	VAR jointtarget CDP_1949 := [[-13.97, 36.67, 4.6, 0, 48.73, -199.13], [9E9, 9E9, 9E9, 9E9, 9E9, 9E9]];
	VAR jointtarget CDP_1950 := [[-13.99, 36.53, 4.84, 0, 48.63, -188.83], [9E9, 9E9, 9E9, 9E9, 9E9, 9E9]];
	VAR jointtarget CDP_1951 := [[-13.98, 36.39, 5.09, 0, 48.52, -178.5], [9E9, 9E9, 9E9, 9E9, 9E9, 9E9]];
	VAR jointtarget CDP_1952 := [[-13.96, 36.25, 5.33, 0, 48.42, -168.15], [9E9, 9E9, 9E9, 9E9, 9E9, 9E9]];
	VAR jointtarget CDP_1953 := [[-13.91, 36.12, 5.55, 0, 48.33, -157.77], [9E9, 9E9, 9E9, 9E9, 9E9, 9E9]];
	VAR jointtarget CDP_1954 := [[-13.84, 36, 5.76, 0, 48.24, -147.38], [9E9, 9E9, 9E9, 9E9, 9E9, 9E9]];
	VAR jointtarget CDP_1955 := [[-13.75, 35.89, 5.94, 0, 48.17, -136.97], [9E9, 9E9, 9E9, 9E9, 9E9, 9E9]];
	VAR jointtarget CDP_1956 := [[-13.64, 35.81, 6.08, 0, 48.11, -126.54], [9E9, 9E9, 9E9, 9E9, 9E9, 9E9]];
	VAR jointtarget CDP_1957 := [[-13.52, 35.74, 6.19, 0, 48.06, -116.09], [9E9, 9E9, 9E9, 9E9, 9E9, 9E9]];
	VAR jointtarget CDP_1958 := [[-13.4, 35.71, 6.26, 0, 48.04, -105.64], [9E9, 9E9, 9E9, 9E9, 9E9, 9E9]];
	VAR jointtarget CDP_1959 := [[-13.27, 35.69, 6.28, 0, 48.03, -95.19], [9E9, 9E9, 9E9, 9E9, 9E9, 9E9]];
	VAR jointtarget CDP_1960 := [[-13.2, 35.69, 6.28, 0, 48.03, -89.96], [9E9, 9E9, 9E9, 9E9, 9E9, 9E9]];
	VAR jointtarget CDP_1961 := [[-13.13, 35.69, 6.28, 0, 48.03, -89.89], [9E9, 9E9, 9E9, 9E9, 9E9, 9E9]];
	VAR jointtarget CDP_1962 := [[-13.06, 35.69, 6.28, 0, 48.03, -89.82], [9E9, 9E9, 9E9, 9E9, 9E9, 9E9]];
	VAR jointtarget CDP_1963 := [[-12.99, 35.69, 6.28, 0, 48.03, -89.75], [9E9, 9E9, 9E9, 9E9, 9E9, 9E9]];
	VAR jointtarget CDP_1964 := [[-12.93, 35.69, 6.28, 0, 48.03, -89.69], [9E9, 9E9, 9E9, 9E9, 9E9, 9E9]];
	VAR jointtarget CDP_1965 := [[-12.86, 35.69, 6.28, 0, 48.03, -89.62], [9E9, 9E9, 9E9, 9E9, 9E9, 9E9]];
	VAR jointtarget CDP_1966 := [[-12.79, 35.69, 6.28, 0, 48.03, -89.55], [9E9, 9E9, 9E9, 9E9, 9E9, 9E9]];
	VAR jointtarget CDP_1967 := [[-12.72, 35.69, 6.28, 0, 48.03, -89.48], [9E9, 9E9, 9E9, 9E9, 9E9, 9E9]];
	VAR jointtarget CDP_1968 := [[-12.65, 35.69, 6.27, 0, 48.03, -89.41], [9E9, 9E9, 9E9, 9E9, 9E9, 9E9]];
	VAR jointtarget CDP_1969 := [[-12.59, 35.69, 6.27, 0, 48.04, -89.35], [9E9, 9E9, 9E9, 9E9, 9E9, 9E9]];
	VAR jointtarget CDP_1970 := [[-12.52, 35.69, 6.27, 0, 48.04, -89.28], [9E9, 9E9, 9E9, 9E9, 9E9, 9E9]];
	VAR jointtarget CDP_1971 := [[-12.45, 35.69, 6.27, 0, 48.04, -89.21], [9E9, 9E9, 9E9, 9E9, 9E9, 9E9]];
	VAR jointtarget CDP_1972 := [[-12.38, 35.69, 6.27, 0, 48.04, -89.14], [9E9, 9E9, 9E9, 9E9, 9E9, 9E9]];
	VAR jointtarget CDP_1973 := [[-12.32, 35.69, 6.27, 0, 48.04, -89.07], [9E9, 9E9, 9E9, 9E9, 9E9, 9E9]];
	VAR jointtarget CDP_1974 := [[-12.25, 35.69, 6.26, 0, 48.04, -89.01], [9E9, 9E9, 9E9, 9E9, 9E9, 9E9]];
	VAR jointtarget CDP_1975 := [[-12.18, 35.69, 6.26, 0, 48.04, -88.94], [9E9, 9E9, 9E9, 9E9, 9E9, 9E9]];
	VAR jointtarget CDP_1976 := [[-12.11, 35.7, 6.26, 0, 48.05, -88.87], [9E9, 9E9, 9E9, 9E9, 9E9, 9E9]];
	VAR jointtarget CDP_1977 := [[-12.04, 35.7, 6.26, 0, 48.05, -88.8], [9E9, 9E9, 9E9, 9E9, 9E9, 9E9]];
	VAR jointtarget CDP_1978 := [[-11.98, 35.7, 6.25, 0, 48.05, -88.74], [9E9, 9E9, 9E9, 9E9, 9E9, 9E9]];
	VAR jointtarget CDP_1979 := [[-11.91, 35.7, 6.25, 0, 48.05, -88.67], [9E9, 9E9, 9E9, 9E9, 9E9, 9E9]];
	VAR jointtarget CDP_1980 := [[-11.89, 35.7, 6.25, 0, 48.05, -88.98], [9E9, 9E9, 9E9, 9E9, 9E9, 9E9]];
	VAR jointtarget CDP_1981 := [[-11.87, 35.7, 6.25, 0, 48.05, -89.63], [9E9, 9E9, 9E9, 9E9, 9E9, 9E9]];
	VAR jointtarget CDP_1982 := [[-11.86, 35.7, 6.25, 0, 48.05, -90.27], [9E9, 9E9, 9E9, 9E9, 9E9, 9E9]];
	VAR jointtarget CDP_1983 := [[-11.84, 35.7, 6.25, 0, 48.05, -90.92], [9E9, 9E9, 9E9, 9E9, 9E9, 9E9]];
	VAR jointtarget CDP_1984 := [[-11.82, 35.7, 6.25, 0, 48.05, -91.56], [9E9, 9E9, 9E9, 9E9, 9E9, 9E9]];
	VAR jointtarget CDP_1985 := [[-11.81, 35.7, 6.25, 0, 48.05, -92.21], [9E9, 9E9, 9E9, 9E9, 9E9, 9E9]];
	VAR jointtarget CDP_1986 := [[-11.79, 35.7, 6.25, 0, 48.05, -92.85], [9E9, 9E9, 9E9, 9E9, 9E9, 9E9]];
	VAR jointtarget CDP_1987 := [[-11.77, 35.69, 6.25, 0, 48.05, -93.5], [9E9, 9E9, 9E9, 9E9, 9E9, 9E9]];
	VAR jointtarget CDP_1988 := [[-11.76, 35.69, 6.26, 0, 48.05, -94.14], [9E9, 9E9, 9E9, 9E9, 9E9, 9E9]];
	VAR jointtarget CDP_1989 := [[-11.74, 35.69, 6.26, 0, 48.05, -94.79], [9E9, 9E9, 9E9, 9E9, 9E9, 9E9]];
	VAR jointtarget CDP_1990 := [[-11.72, 35.69, 6.26, 0, 48.05, -95.43], [9E9, 9E9, 9E9, 9E9, 9E9, 9E9]];
	VAR jointtarget CDP_1991 := [[-11.71, 35.69, 6.27, 0, 48.05, -96.08], [9E9, 9E9, 9E9, 9E9, 9E9, 9E9]];
	VAR jointtarget CDP_1992 := [[-11.69, 35.69, 6.27, 0, 48.05, -96.72], [9E9, 9E9, 9E9, 9E9, 9E9, 9E9]];
	VAR jointtarget CDP_1993 := [[-11.67, 35.68, 6.27, 0, 48.04, -97.37], [9E9, 9E9, 9E9, 9E9, 9E9, 9E9]];
	VAR jointtarget CDP_1994 := [[-11.66, 35.68, 6.28, 0, 48.04, -98.01], [9E9, 9E9, 9E9, 9E9, 9E9, 9E9]];
	VAR jointtarget CDP_1995 := [[-11.64, 35.68, 6.28, 0, 48.04, -98.66], [9E9, 9E9, 9E9, 9E9, 9E9, 9E9]];
	VAR jointtarget CDP_1996 := [[-11.62, 35.67, 6.29, 0, 48.04, -99.31], [9E9, 9E9, 9E9, 9E9, 9E9, 9E9]];
	VAR jointtarget CDP_1997 := [[-11.61, 35.67, 6.29, 0, 48.04, -99.95], [9E9, 9E9, 9E9, 9E9, 9E9, 9E9]];
	VAR jointtarget CDP_1998 := [[-11.59, 35.67, 6.3, 0, 48.03, -100.6], [9E9, 9E9, 9E9, 9E9, 9E9, 9E9]];
	VAR jointtarget CDP_1999 := [[-11.57, 35.66, 6.3, 0, 48.03, -101.24], [9E9, 9E9, 9E9, 9E9, 9E9, 9E9]];
	VAR jointtarget CDP_2000 := [[-10.48, 35.44, 6.7, 0, 47.87, -100.48], [9E9, 9E9, 9E9, 9E9, 9E9, 9E9]];
	VAR jointtarget CDP_2001 := [[-9.38, 35.23, 7.05, 0, 47.72, -99.38], [9E9, 9E9, 9E9, 9E9, 9E9, 9E9]];
	VAR jointtarget CDP_2002 := [[-8.27, 35.05, 7.36, 0, 47.59, -98.27], [9E9, 9E9, 9E9, 9E9, 9E9, 9E9]];
	VAR jointtarget CDP_2003 := [[-7.15, 34.89, 7.63, 0, 47.48, -97.15], [9E9, 9E9, 9E9, 9E9, 9E9, 9E9]];
	VAR jointtarget CDP_2004 := [[-6.03, 34.75, 7.87, 0, 47.38, -96.03], [9E9, 9E9, 9E9, 9E9, 9E9, 9E9]];
	VAR jointtarget CDP_2005 := [[-4.9, 34.64, 8.06, 0, 47.31, -94.9], [9E9, 9E9, 9E9, 9E9, 9E9, 9E9]];
	VAR jointtarget CDP_2006 := [[-3.77, 34.55, 8.21, 0, 47.24, -93.77], [9E9, 9E9, 9E9, 9E9, 9E9, 9E9]];
	VAR jointtarget CDP_2007 := [[-2.64, 34.48, 8.32, 0, 47.2, -92.64], [9E9, 9E9, 9E9, 9E9, 9E9, 9E9]];
	VAR jointtarget CDP_2008 := [[-1.51, 34.44, 8.4, 0, 47.17, -91.51], [9E9, 9E9, 9E9, 9E9, 9E9, 9E9]];
	VAR jointtarget CDP_2009 := [[-0.37, 34.42, 8.43, 0, 47.15, -90.37], [9E9, 9E9, 9E9, 9E9, 9E9, 9E9]];
	VAR jointtarget CDP_2010 := [[0.76, 34.42, 8.42, 0, 47.15, -89.24], [9E9, 9E9, 9E9, 9E9, 9E9, 9E9]];
	VAR jointtarget CDP_2011 := [[1.9, 34.45, 8.38, 0, 47.17, -88.1], [9E9, 9E9, 9E9, 9E9, 9E9, 9E9]];
	VAR jointtarget CDP_2012 := [[3.03, 34.5, 8.29, 0, 47.21, -86.97], [9E9, 9E9, 9E9, 9E9, 9E9, 9E9]];
	VAR jointtarget CDP_2013 := [[4.16, 34.57, 8.16, 0, 47.26, -85.84], [9E9, 9E9, 9E9, 9E9, 9E9, 9E9]];
	VAR jointtarget CDP_2014 := [[5.29, 34.67, 8, 0, 47.33, -84.71], [9E9, 9E9, 9E9, 9E9, 9E9, 9E9]];
	VAR jointtarget CDP_2015 := [[6.42, 34.79, 7.79, 0, 47.42, -83.58], [9E9, 9E9, 9E9, 9E9, 9E9, 9E9]];
	VAR jointtarget CDP_2016 := [[7.54, 34.94, 7.54, 0, 47.52, -82.46], [9E9, 9E9, 9E9, 9E9, 9E9, 9E9]];
	VAR jointtarget CDP_2017 := [[8.65, 35.11, 7.26, 0, 47.64, -81.35], [9E9, 9E9, 9E9, 9E9, 9E9, 9E9]];
	VAR jointtarget CDP_2018 := [[9.76, 35.3, 6.93, 0, 47.77, -80.24], [9E9, 9E9, 9E9, 9E9, 9E9, 9E9]];
	VAR jointtarget CDP_2019 := [[10.86, 35.51, 6.57, 0, 47.92, -79.14], [9E9, 9E9, 9E9, 9E9, 9E9, 9E9]];
	VAR jointtarget CDP_2020 := [[10.87, 35.52, 6.56, 0, 47.92, -79.46], [9E9, 9E9, 9E9, 9E9, 9E9, 9E9]];
	VAR jointtarget CDP_2021 := [[10.89, 35.52, 6.55, 0, 47.93, -80.1], [9E9, 9E9, 9E9, 9E9, 9E9, 9E9]];
	VAR jointtarget CDP_2022 := [[10.91, 35.52, 6.55, 0, 47.93, -80.75], [9E9, 9E9, 9E9, 9E9, 9E9, 9E9]];
	VAR jointtarget CDP_2023 := [[10.92, 35.52, 6.55, 0, 47.93, -81.39], [9E9, 9E9, 9E9, 9E9, 9E9, 9E9]];
	VAR jointtarget CDP_2024 := [[10.94, 35.53, 6.54, 0, 47.93, -82.04], [9E9, 9E9, 9E9, 9E9, 9E9, 9E9]];
	VAR jointtarget CDP_2025 := [[10.96, 35.53, 6.54, 0, 47.93, -82.68], [9E9, 9E9, 9E9, 9E9, 9E9, 9E9]];
	VAR jointtarget CDP_2026 := [[10.97, 35.53, 6.53, 0, 47.94, -83.33], [9E9, 9E9, 9E9, 9E9, 9E9, 9E9]];
	VAR jointtarget CDP_2027 := [[10.99, 35.53, 6.53, 0, 47.94, -83.97], [9E9, 9E9, 9E9, 9E9, 9E9, 9E9]];
	VAR jointtarget CDP_2028 := [[11.01, 35.53, 6.53, 0, 47.94, -84.62], [9E9, 9E9, 9E9, 9E9, 9E9, 9E9]];
	VAR jointtarget CDP_2029 := [[11.02, 35.54, 6.52, 0, 47.94, -85.27], [9E9, 9E9, 9E9, 9E9, 9E9, 9E9]];
	VAR jointtarget CDP_2030 := [[11.04, 35.54, 6.52, 0, 47.94, -85.91], [9E9, 9E9, 9E9, 9E9, 9E9, 9E9]];
	VAR jointtarget CDP_2031 := [[11.06, 35.54, 6.52, 0, 47.94, -86.56], [9E9, 9E9, 9E9, 9E9, 9E9, 9E9]];
	VAR jointtarget CDP_2032 := [[11.07, 35.54, 6.52, 0, 47.94, -87.2], [9E9, 9E9, 9E9, 9E9, 9E9, 9E9]];
	VAR jointtarget CDP_2033 := [[11.09, 35.54, 6.52, 0, 47.94, -87.85], [9E9, 9E9, 9E9, 9E9, 9E9, 9E9]];
	VAR jointtarget CDP_2034 := [[11.11, 35.54, 6.52, 0, 47.94, -88.49], [9E9, 9E9, 9E9, 9E9, 9E9, 9E9]];
	VAR jointtarget CDP_2035 := [[11.13, 35.54, 6.52, 0, 47.94, -89.14], [9E9, 9E9, 9E9, 9E9, 9E9, 9E9]];
	VAR jointtarget CDP_2036 := [[11.14, 35.54, 6.52, 0, 47.94, -89.78], [9E9, 9E9, 9E9, 9E9, 9E9, 9E9]];
	VAR jointtarget CDP_2037 := [[11.16, 35.54, 6.52, 0, 47.94, -90.43], [9E9, 9E9, 9E9, 9E9, 9E9, 9E9]];
	VAR jointtarget CDP_2038 := [[11.18, 35.54, 6.52, 0, 47.94, -91.07], [9E9, 9E9, 9E9, 9E9, 9E9, 9E9]];
	VAR jointtarget CDP_2039 := [[11.19, 35.54, 6.52, 0, 47.94, -91.72], [9E9, 9E9, 9E9, 9E9, 9E9, 9E9]];
	VAR jointtarget CDP_2040 := [[11.26, 35.54, 6.52, 0, 47.94, -91.98], [9E9, 9E9, 9E9, 9E9, 9E9, 9E9]];
	VAR jointtarget CDP_2041 := [[11.33, 35.53, 6.53, 0, 47.94, -91.91], [9E9, 9E9, 9E9, 9E9, 9E9, 9E9]];
	VAR jointtarget CDP_2042 := [[11.4, 35.53, 6.53, 0, 47.94, -91.84], [9E9, 9E9, 9E9, 9E9, 9E9, 9E9]];
	VAR jointtarget CDP_2043 := [[11.47, 35.53, 6.53, 0, 47.94, -91.78], [9E9, 9E9, 9E9, 9E9, 9E9, 9E9]];
	VAR jointtarget CDP_2044 := [[11.53, 35.53, 6.54, 0, 47.93, -91.71], [9E9, 9E9, 9E9, 9E9, 9E9, 9E9]];
	VAR jointtarget CDP_2045 := [[11.6, 35.53, 6.54, 0, 47.93, -91.64], [9E9, 9E9, 9E9, 9E9, 9E9, 9E9]];
	VAR jointtarget CDP_2046 := [[11.67, 35.52, 6.55, 0, 47.93, -91.57], [9E9, 9E9, 9E9, 9E9, 9E9, 9E9]];
	VAR jointtarget CDP_2047 := [[11.74, 35.52, 6.55, 0, 47.93, -91.5], [9E9, 9E9, 9E9, 9E9, 9E9, 9E9]];
	VAR jointtarget CDP_2048 := [[11.81, 35.52, 6.55, 0, 47.93, -91.44], [9E9, 9E9, 9E9, 9E9, 9E9, 9E9]];
	VAR jointtarget CDP_2049 := [[11.87, 35.52, 6.56, 0, 47.93, -91.37], [9E9, 9E9, 9E9, 9E9, 9E9, 9E9]];
	VAR jointtarget CDP_2050 := [[11.94, 35.52, 6.56, 0, 47.93, -91.3], [9E9, 9E9, 9E9, 9E9, 9E9, 9E9]];
	VAR jointtarget CDP_2051 := [[12.01, 35.51, 6.56, 0, 47.92, -91.23], [9E9, 9E9, 9E9, 9E9, 9E9, 9E9]];
	VAR jointtarget CDP_2052 := [[12.08, 35.51, 6.56, 0, 47.92, -91.16], [9E9, 9E9, 9E9, 9E9, 9E9, 9E9]];
	VAR jointtarget CDP_2053 := [[12.15, 35.51, 6.57, 0, 47.92, -91.09], [9E9, 9E9, 9E9, 9E9, 9E9, 9E9]];
	VAR jointtarget CDP_2054 := [[12.21, 35.51, 6.57, 0, 47.92, -91.03], [9E9, 9E9, 9E9, 9E9, 9E9, 9E9]];
	VAR jointtarget CDP_2055 := [[12.28, 35.51, 6.57, 0, 47.92, -90.96], [9E9, 9E9, 9E9, 9E9, 9E9, 9E9]];
	VAR jointtarget CDP_2056 := [[12.35, 35.51, 6.57, 0, 47.92, -90.89], [9E9, 9E9, 9E9, 9E9, 9E9, 9E9]];
	VAR jointtarget CDP_2057 := [[12.42, 35.51, 6.57, 0, 47.92, -90.82], [9E9, 9E9, 9E9, 9E9, 9E9, 9E9]];
	VAR jointtarget CDP_2058 := [[12.49, 35.51, 6.58, 0, 47.92, -90.75], [9E9, 9E9, 9E9, 9E9, 9E9, 9E9]];
	VAR jointtarget CDP_2059 := [[12.55, 35.5, 6.58, 0, 47.92, -90.69], [9E9, 9E9, 9E9, 9E9, 9E9, 9E9]];
	VAR jointtarget CDP_2060 := [[12.69, 35.52, 6.56, 0, 47.93, -85.39], [9E9, 9E9, 9E9, 9E9, 9E9, 9E9]];
	VAR jointtarget CDP_2061 := [[12.81, 35.55, 6.5, 0, 47.95, -74.94], [9E9, 9E9, 9E9, 9E9, 9E9, 9E9]];
	VAR jointtarget CDP_2062 := [[12.93, 35.61, 6.39, 0, 47.99, -64.5], [9E9, 9E9, 9E9, 9E9, 9E9, 9E9]];
	VAR jointtarget CDP_2063 := [[13.04, 35.7, 6.25, 0, 48.05, -54.07], [9E9, 9E9, 9E9, 9E9, 9E9, 9E9]];
	VAR jointtarget CDP_2064 := [[13.13, 35.8, 6.07, 0, 48.13, -43.65], [9E9, 9E9, 9E9, 9E9, 9E9, 9E9]];
	VAR jointtarget CDP_2065 := [[13.2, 35.92, 5.87, 0, 48.21, -33.25], [9E9, 9E9, 9E9, 9E9, 9E9, 9E9]];
	VAR jointtarget CDP_2066 := [[13.25, 36.05, 5.64, 0, 48.31, -22.88], [9E9, 9E9, 9E9, 9E9, 9E9, 9E9]];
	VAR jointtarget CDP_2067 := [[13.28, 36.19, 5.4, 0, 48.41, -12.53], [9E9, 9E9, 9E9, 9E9, 9E9, 9E9]];
	VAR jointtarget CDP_2068 := [[13.29, 36.33, 5.16, 0, 48.51, -2.2], [9E9, 9E9, 9E9, 9E9, 9E9, 9E9]];
	VAR jointtarget CDP_2069 := [[13.27, 36.47, 4.92, 0, 48.61, 8.11], [9E9, 9E9, 9E9, 9E9, 9E9, 9E9]];
	VAR jointtarget CDP_2070 := [[13.23, 36.61, 4.68, 0, 48.71, 18.39], [9E9, 9E9, 9E9, 9E9, 9E9, 9E9]];
	VAR jointtarget CDP_2071 := [[13.17, 36.74, 4.47, 0, 48.8, 28.65], [9E9, 9E9, 9E9, 9E9, 9E9, 9E9]];
	VAR jointtarget CDP_2072 := [[13.08, 36.85, 4.27, 0, 48.88, 38.9], [9E9, 9E9, 9E9, 9E9, 9E9, 9E9]];
	VAR jointtarget CDP_2073 := [[12.99, 36.94, 4.11, 0, 48.95, 49.12], [9E9, 9E9, 9E9, 9E9, 9E9, 9E9]];
	VAR jointtarget CDP_2074 := [[12.88, 37.02, 3.98, 0, 49, 59.33], [9E9, 9E9, 9E9, 9E9, 9E9, 9E9]];
	VAR jointtarget CDP_2075 := [[12.75, 37.07, 3.9, 0, 49.04, 69.54], [9E9, 9E9, 9E9, 9E9, 9E9, 9E9]];
	VAR jointtarget CDP_2076 := [[12.63, 37.09, 3.85, 0, 49.05, 79.73], [9E9, 9E9, 9E9, 9E9, 9E9, 9E9]];
	VAR jointtarget CDP_2077 := [[12.5, 37.09, 3.85, 0, 49.05, 89.93], [9E9, 9E9, 9E9, 9E9, 9E9, 9E9]];
	VAR jointtarget CDP_2078 := [[12.37, 37.07, 3.9, 0, 49.04, 100.13], [9E9, 9E9, 9E9, 9E9, 9E9, 9E9]];
	VAR jointtarget CDP_2079 := [[12.25, 37.02, 3.98, 0, 49, 110.33], [9E9, 9E9, 9E9, 9E9, 9E9, 9E9]];
	VAR jointtarget CDP_2080 := [[12.19, 36.98, 4.04, 0, 48.98, 115.43], [9E9, 9E9, 9E9, 9E9, 9E9, 9E9]];
	VAR jointtarget CDP_2081 := [[12.13, 36.95, 4.09, 0, 48.95, 115.37], [9E9, 9E9, 9E9, 9E9, 9E9, 9E9]];
	VAR jointtarget CDP_2082 := [[12.07, 36.92, 4.15, 0, 48.93, 115.31], [9E9, 9E9, 9E9, 9E9, 9E9, 9E9]];
	VAR jointtarget CDP_2083 := [[12.01, 36.89, 4.2, 0, 48.91, 115.25], [9E9, 9E9, 9E9, 9E9, 9E9, 9E9]];
	VAR jointtarget CDP_2084 := [[11.95, 36.86, 4.26, 0, 48.89, 115.19], [9E9, 9E9, 9E9, 9E9, 9E9, 9E9]];
	VAR jointtarget CDP_2085 := [[11.89, 36.83, 4.31, 0, 48.86, 115.13], [9E9, 9E9, 9E9, 9E9, 9E9, 9E9]];
	VAR jointtarget CDP_2086 := [[11.83, 36.79, 4.37, 0, 48.84, 115.07], [9E9, 9E9, 9E9, 9E9, 9E9, 9E9]];
	VAR jointtarget CDP_2087 := [[11.77, 36.76, 4.42, 0, 48.82, 115.01], [9E9, 9E9, 9E9, 9E9, 9E9, 9E9]];
	VAR jointtarget CDP_2088 := [[11.71, 36.73, 4.47, 0, 48.8, 114.95], [9E9, 9E9, 9E9, 9E9, 9E9, 9E9]];
	VAR jointtarget CDP_2089 := [[11.65, 36.7, 4.53, 0, 48.77, 114.89], [9E9, 9E9, 9E9, 9E9, 9E9, 9E9]];
	VAR jointtarget CDP_2090 := [[11.59, 36.67, 4.58, 0, 48.75, 114.83], [9E9, 9E9, 9E9, 9E9, 9E9, 9E9]];
	VAR jointtarget CDP_2091 := [[11.53, 36.64, 4.63, 0, 48.73, 114.77], [9E9, 9E9, 9E9, 9E9, 9E9, 9E9]];
	VAR jointtarget CDP_2092 := [[11.47, 36.61, 4.69, 0, 48.71, 114.71], [9E9, 9E9, 9E9, 9E9, 9E9, 9E9]];
	VAR jointtarget CDP_2093 := [[11.4, 36.58, 4.74, 0, 48.68, 114.64], [9E9, 9E9, 9E9, 9E9, 9E9, 9E9]];
	VAR jointtarget CDP_2094 := [[11.34, 36.55, 4.79, 0, 48.66, 114.58], [9E9, 9E9, 9E9, 9E9, 9E9, 9E9]];
	VAR jointtarget CDP_2095 := [[11.28, 36.52, 4.84, 0, 48.64, 114.52], [9E9, 9E9, 9E9, 9E9, 9E9, 9E9]];
	VAR jointtarget CDP_2096 := [[11.22, 36.49, 4.9, 0, 48.62, 114.46], [9E9, 9E9, 9E9, 9E9, 9E9, 9E9]];
	VAR jointtarget CDP_2097 := [[11.16, 36.46, 4.95, 0, 48.6, 114.4], [9E9, 9E9, 9E9, 9E9, 9E9, 9E9]];
	VAR jointtarget CDP_2098 := [[11.1, 36.42, 5, 0, 48.57, 114.34], [9E9, 9E9, 9E9, 9E9, 9E9, 9E9]];
	VAR jointtarget CDP_2099 := [[11.04, 36.39, 5.05, 0, 48.55, 114.28], [9E9, 9E9, 9E9, 9E9, 9E9, 9E9]];
	VAR jointtarget CDP_2100 := [[11.02, 36.39, 5.07, 0, 48.55, 113.93], [9E9, 9E9, 9E9, 9E9, 9E9, 9E9]];
	VAR jointtarget CDP_2101 := [[11.01, 36.38, 5.08, 0, 48.54, 113.26], [9E9, 9E9, 9E9, 9E9, 9E9, 9E9]];
	VAR jointtarget CDP_2102 := [[10.99, 36.37, 5.09, 0, 48.54, 112.58], [9E9, 9E9, 9E9, 9E9, 9E9, 9E9]];
	VAR jointtarget CDP_2103 := [[10.98, 36.37, 5.1, 0, 48.53, 111.9], [9E9, 9E9, 9E9, 9E9, 9E9, 9E9]];
	VAR jointtarget CDP_2104 := [[10.96, 36.36, 5.11, 0, 48.53, 111.22], [9E9, 9E9, 9E9, 9E9, 9E9, 9E9]];
	VAR jointtarget CDP_2105 := [[10.95, 36.35, 5.12, 0, 48.52, 110.55], [9E9, 9E9, 9E9, 9E9, 9E9, 9E9]];
	VAR jointtarget CDP_2106 := [[10.93, 36.35, 5.14, 0, 48.52, 109.87], [9E9, 9E9, 9E9, 9E9, 9E9, 9E9]];
	VAR jointtarget CDP_2107 := [[10.91, 36.34, 5.15, 0, 48.51, 109.19], [9E9, 9E9, 9E9, 9E9, 9E9, 9E9]];
	VAR jointtarget CDP_2108 := [[10.9, 36.33, 5.16, 0, 48.51, 108.51], [9E9, 9E9, 9E9, 9E9, 9E9, 9E9]];
	VAR jointtarget CDP_2109 := [[10.88, 36.33, 5.17, 0, 48.51, 107.83], [9E9, 9E9, 9E9, 9E9, 9E9, 9E9]];
	VAR jointtarget CDP_2110 := [[10.87, 36.32, 5.17, 0, 48.5, 107.16], [9E9, 9E9, 9E9, 9E9, 9E9, 9E9]];
	VAR jointtarget CDP_2111 := [[10.85, 36.32, 5.18, 0, 48.5, 106.48], [9E9, 9E9, 9E9, 9E9, 9E9, 9E9]];
	VAR jointtarget CDP_2112 := [[10.83, 36.31, 5.19, 0, 48.49, 105.8], [9E9, 9E9, 9E9, 9E9, 9E9, 9E9]];
	VAR jointtarget CDP_2113 := [[10.82, 36.31, 5.2, 0, 48.49, 105.12], [9E9, 9E9, 9E9, 9E9, 9E9, 9E9]];
	VAR jointtarget CDP_2114 := [[10.8, 36.3, 5.21, 0, 48.49, 104.44], [9E9, 9E9, 9E9, 9E9, 9E9, 9E9]];
	VAR jointtarget CDP_2115 := [[10.79, 36.3, 5.22, 0, 48.48, 103.77], [9E9, 9E9, 9E9, 9E9, 9E9, 9E9]];
	VAR jointtarget CDP_2116 := [[10.77, 36.3, 5.22, 0, 48.48, 103.09], [9E9, 9E9, 9E9, 9E9, 9E9, 9E9]];
	VAR jointtarget CDP_2117 := [[10.75, 36.29, 5.23, 0, 48.48, 102.41], [9E9, 9E9, 9E9, 9E9, 9E9, 9E9]];
	VAR jointtarget CDP_2118 := [[10.74, 36.29, 5.24, 0, 48.48, 101.73], [9E9, 9E9, 9E9, 9E9, 9E9, 9E9]];
	VAR jointtarget CDP_2119 := [[10.72, 36.28, 5.24, 0, 48.47, 101.05], [9E9, 9E9, 9E9, 9E9, 9E9, 9E9]];
	VAR jointtarget CDP_2120 := [[9.64, 36.07, 5.6, 0, 48.32, 99.64], [9E9, 9E9, 9E9, 9E9, 9E9, 9E9]];
	VAR jointtarget CDP_2121 := [[8.56, 35.89, 5.93, 0, 48.19, 98.56], [9E9, 9E9, 9E9, 9E9, 9E9, 9E9]];
	VAR jointtarget CDP_2122 := [[7.47, 35.72, 6.21, 0, 48.07, 97.47], [9E9, 9E9, 9E9, 9E9, 9E9, 9E9]];
	VAR jointtarget CDP_2123 := [[6.38, 35.58, 6.46, 0, 47.97, 96.38], [9E9, 9E9, 9E9, 9E9, 9E9, 9E9]];
	VAR jointtarget CDP_2124 := [[5.28, 35.46, 6.66, 0, 47.88, 95.28], [9E9, 9E9, 9E9, 9E9, 9E9, 9E9]];
	VAR jointtarget CDP_2125 := [[4.17, 35.36, 6.83, 0, 47.81, 94.17], [9E9, 9E9, 9E9, 9E9, 9E9, 9E9]];
	VAR jointtarget CDP_2126 := [[3.07, 35.28, 6.96, 0, 47.76, 93.07], [9E9, 9E9, 9E9, 9E9, 9E9, 9E9]];
	VAR jointtarget CDP_2127 := [[1.96, 35.23, 7.04, 0, 47.72, 91.96], [9E9, 9E9, 9E9, 9E9, 9E9, 9E9]];
	VAR jointtarget CDP_2128 := [[0.85, 35.2, 7.09, 0, 47.7, 90.85], [9E9, 9E9, 9E9, 9E9, 9E9, 9E9]];
	VAR jointtarget CDP_2129 := [[-0.26, 35.2, 7.1, 0, 47.7, 89.74], [9E9, 9E9, 9E9, 9E9, 9E9, 9E9]];
	VAR jointtarget CDP_2130 := [[-1.37, 35.21, 7.08, 0, 47.71, 88.63], [9E9, 9E9, 9E9, 9E9, 9E9, 9E9]];
	VAR jointtarget CDP_2131 := [[-2.48, 35.25, 7.01, 0, 47.74, 87.52], [9E9, 9E9, 9E9, 9E9, 9E9, 9E9]];
	VAR jointtarget CDP_2132 := [[-3.59, 35.32, 6.9, 0, 47.78, 86.41], [9E9, 9E9, 9E9, 9E9, 9E9, 9E9]];
	VAR jointtarget CDP_2133 := [[-4.7, 35.4, 6.75, 0, 47.84, 85.3], [9E9, 9E9, 9E9, 9E9, 9E9, 9E9]];
	VAR jointtarget CDP_2134 := [[-5.8, 35.51, 6.57, 0, 47.92, 84.2], [9E9, 9E9, 9E9, 9E9, 9E9, 9E9]];
	VAR jointtarget CDP_2135 := [[-6.9, 35.64, 6.34, 0, 48.01, 83.1], [9E9, 9E9, 9E9, 9E9, 9E9, 9E9]];
	VAR jointtarget CDP_2136 := [[-7.99, 35.8, 6.08, 0, 48.12, 82.01], [9E9, 9E9, 9E9, 9E9, 9E9, 9E9]];
	VAR jointtarget CDP_2137 := [[-9.08, 35.97, 5.78, 0, 48.25, 80.92], [9E9, 9E9, 9E9, 9E9, 9E9, 9E9]];
	VAR jointtarget CDP_2138 := [[-10.16, 36.17, 5.44, 0, 48.39, 79.84], [9E9, 9E9, 9E9, 9E9, 9E9, 9E9]];
	VAR jointtarget CDP_2139 := [[-11.23, 36.39, 5.06, 0, 48.55, 78.77], [9E9, 9E9, 9E9, 9E9, 9E9, 9E9]];
	VAR jointtarget CDP_2140 := [[-11.28, 36.4, 5.04, 0, 48.56, 79.81], [9E9, 9E9, 9E9, 9E9, 9E9, 9E9]];
	VAR jointtarget CDP_2141 := [[-11.34, 36.41, 5.02, 0, 48.56, 81.95], [9E9, 9E9, 9E9, 9E9, 9E9, 9E9]];
	VAR jointtarget CDP_2142 := [[-11.39, 36.42, 5.01, 0, 48.57, 84.09], [9E9, 9E9, 9E9, 9E9, 9E9, 9E9]];
	VAR jointtarget CDP_2143 := [[-11.45, 36.42, 5.01, 0, 48.57, 86.23], [9E9, 9E9, 9E9, 9E9, 9E9, 9E9]];
	VAR jointtarget CDP_2144 := [[-11.5, 36.42, 5, 0, 48.57, 88.37], [9E9, 9E9, 9E9, 9E9, 9E9, 9E9]];
	VAR jointtarget CDP_2145 := [[-11.56, 36.42, 5, 0, 48.57, 90.51], [9E9, 9E9, 9E9, 9E9, 9E9, 9E9]];
	VAR jointtarget CDP_2146 := [[-11.61, 36.42, 5.01, 0, 48.57, 92.65], [9E9, 9E9, 9E9, 9E9, 9E9, 9E9]];
	VAR jointtarget CDP_2147 := [[-11.67, 36.42, 5.02, 0, 48.57, 94.78], [9E9, 9E9, 9E9, 9E9, 9E9, 9E9]];
	VAR jointtarget CDP_2148 := [[-11.72, 36.41, 5.03, 0, 48.56, 96.92], [9E9, 9E9, 9E9, 9E9, 9E9, 9E9]];
	VAR jointtarget CDP_2149 := [[-11.78, 36.4, 5.05, 0, 48.55, 99.06], [9E9, 9E9, 9E9, 9E9, 9E9, 9E9]];
	VAR jointtarget CDP_2150 := [[-11.83, 36.39, 5.07, 0, 48.55, 101.2], [9E9, 9E9, 9E9, 9E9, 9E9, 9E9]];
	VAR jointtarget CDP_2151 := [[-11.89, 36.37, 5.09, 0, 48.54, 103.34], [9E9, 9E9, 9E9, 9E9, 9E9, 9E9]];
	VAR jointtarget CDP_2152 := [[-11.94, 36.36, 5.12, 0, 48.52, 105.48], [9E9, 9E9, 9E9, 9E9, 9E9, 9E9]];
	VAR jointtarget CDP_2153 := [[-11.99, 36.34, 5.15, 0, 48.51, 107.63], [9E9, 9E9, 9E9, 9E9, 9E9, 9E9]];
	VAR jointtarget CDP_2154 := [[-12.04, 36.32, 5.19, 0, 48.5, 109.77], [9E9, 9E9, 9E9, 9E9, 9E9, 9E9]];
	VAR jointtarget CDP_2155 := [[-12.09, 36.3, 5.22, 0, 48.48, 111.91], [9E9, 9E9, 9E9, 9E9, 9E9, 9E9]];
	VAR jointtarget CDP_2156 := [[-12.15, 36.27, 5.27, 0, 48.46, 114.05], [9E9, 9E9, 9E9, 9E9, 9E9, 9E9]];
	VAR jointtarget CDP_2157 := [[-12.19, 36.24, 5.31, 0, 48.44, 116.2], [9E9, 9E9, 9E9, 9E9, 9E9, 9E9]];
	VAR jointtarget CDP_2158 := [[-12.24, 36.22, 5.36, 0, 48.42, 118.34], [9E9, 9E9, 9E9, 9E9, 9E9, 9E9]];
	VAR jointtarget CDP_2159 := [[-12.29, 36.18, 5.41, 0, 48.4, 120.49], [9E9, 9E9, 9E9, 9E9, 9E9, 9E9]];
	VAR jointtarget CDP_2160 := [[-12.32, 36.17, 5.45, 0, 48.39, 121.56], [9E9, 9E9, 9E9, 9E9, 9E9, 9E9]];
	VAR jointtarget CDP_2161 := [[-12.35, 36.15, 5.48, 0, 48.37, 121.53], [9E9, 9E9, 9E9, 9E9, 9E9, 9E9]];
	VAR jointtarget CDP_2162 := [[-12.38, 36.13, 5.51, 0, 48.36, 121.5], [9E9, 9E9, 9E9, 9E9, 9E9, 9E9]];
	VAR jointtarget CDP_2163 := [[-12.41, 36.11, 5.54, 0, 48.35, 121.47], [9E9, 9E9, 9E9, 9E9, 9E9, 9E9]];
	VAR jointtarget CDP_2164 := [[-12.43, 36.09, 5.58, 0, 48.33, 121.44], [9E9, 9E9, 9E9, 9E9, 9E9, 9E9]];
	VAR jointtarget CDP_2165 := [[-12.46, 36.07, 5.61, 0, 48.32, 121.41], [9E9, 9E9, 9E9, 9E9, 9E9, 9E9]];
	VAR jointtarget CDP_2166 := [[-12.49, 36.05, 5.64, 0, 48.31, 121.39], [9E9, 9E9, 9E9, 9E9, 9E9, 9E9]];
	VAR jointtarget CDP_2167 := [[-12.52, 36.03, 5.68, 0, 48.29, 121.36], [9E9, 9E9, 9E9, 9E9, 9E9, 9E9]];
	VAR jointtarget CDP_2168 := [[-12.55, 36.01, 5.71, 0, 48.28, 121.33], [9E9, 9E9, 9E9, 9E9, 9E9, 9E9]];
	VAR jointtarget CDP_2169 := [[-12.58, 35.99, 5.74, 0, 48.27, 121.3], [9E9, 9E9, 9E9, 9E9, 9E9, 9E9]];
	VAR jointtarget CDP_2170 := [[-12.61, 35.98, 5.77, 0, 48.25, 121.27], [9E9, 9E9, 9E9, 9E9, 9E9, 9E9]];
	VAR jointtarget CDP_2171 := [[-12.63, 35.96, 5.81, 0, 48.24, 121.24], [9E9, 9E9, 9E9, 9E9, 9E9, 9E9]];
	VAR jointtarget CDP_2172 := [[-12.66, 35.94, 5.84, 0, 48.23, 121.21], [9E9, 9E9, 9E9, 9E9, 9E9, 9E9]];
	VAR jointtarget CDP_2173 := [[-12.69, 35.92, 5.87, 0, 48.21, 121.18], [9E9, 9E9, 9E9, 9E9, 9E9, 9E9]];
	VAR jointtarget CDP_2174 := [[-12.72, 35.9, 5.9, 0, 48.2, 121.16], [9E9, 9E9, 9E9, 9E9, 9E9, 9E9]];
	VAR jointtarget CDP_2175 := [[-12.75, 35.88, 5.93, 0, 48.18, 121.13], [9E9, 9E9, 9E9, 9E9, 9E9, 9E9]];
	VAR jointtarget CDP_2176 := [[-12.78, 35.86, 5.97, 0, 48.17, 121.1], [9E9, 9E9, 9E9, 9E9, 9E9, 9E9]];
	VAR jointtarget CDP_2177 := [[-12.81, 35.84, 6, 0, 48.16, 121.07], [9E9, 9E9, 9E9, 9E9, 9E9, 9E9]];
	VAR jointtarget CDP_2178 := [[-12.84, 35.82, 6.03, 0, 48.14, 121.04], [9E9, 9E9, 9E9, 9E9, 9E9, 9E9]];
	VAR jointtarget CDP_2179 := [[-12.86, 35.81, 6.06, 0, 48.13, 121.01], [9E9, 9E9, 9E9, 9E9, 9E9, 9E9]];
	VAR jointtarget CDP_2180 := [[-13.02, 35.73, 6.19, 0, 48.08, 114.17], [9E9, 9E9, 9E9, 9E9, 9E9, 9E9]];
	VAR jointtarget CDP_2181 := [[-13.18, 35.7, 6.24, 0, 48.06, 100.62], [9E9, 9E9, 9E9, 9E9, 9E9, 9E9]];
	VAR jointtarget CDP_2182 := [[-13.34, 35.71, 6.23, 0, 48.06, 87.07], [9E9, 9E9, 9E9, 9E9, 9E9, 9E9]];
	VAR jointtarget CDP_2183 := [[-13.5, 35.76, 6.14, 0, 48.1, 73.52], [9E9, 9E9, 9E9, 9E9, 9E9, 9E9]];
	VAR jointtarget CDP_2184 := [[-13.64, 35.85, 5.99, 0, 48.16, 59.99], [9E9, 9E9, 9E9, 9E9, 9E9, 9E9]];
	VAR jointtarget CDP_2185 := [[-13.76, 35.97, 5.78, 0, 48.25, 46.48], [9E9, 9E9, 9E9, 9E9, 9E9, 9E9]];
	VAR jointtarget CDP_2186 := [[-13.85, 36.12, 5.53, 0, 48.36, 33.01], [9E9, 9E9, 9E9, 9E9, 9E9, 9E9]];
	VAR jointtarget CDP_2187 := [[-13.91, 36.29, 5.24, 0, 48.48, 19.56], [9E9, 9E9, 9E9, 9E9, 9E9, 9E9]];
	VAR jointtarget CDP_2188 := [[-13.92, 36.47, 4.93, 0, 48.6, 6.16], [9E9, 9E9, 9E9, 9E9, 9E9, 9E9]];
	VAR jointtarget CDP_2189 := [[-13.9, 36.64, 4.63, 0, 48.73, -7.21], [9E9, 9E9, 9E9, 9E9, 9E9, 9E9]];
	VAR jointtarget CDP_2190 := [[-13.85, 36.81, 4.34, 0, 48.85, -20.54], [9E9, 9E9, 9E9, 9E9, 9E9, 9E9]];
	VAR jointtarget CDP_2191 := [[-13.76, 36.96, 4.08, 0, 48.96, -33.84], [9E9, 9E9, 9E9, 9E9, 9E9, 9E9]];
	VAR jointtarget CDP_2192 := [[-13.64, 37.08, 3.87, 0, 49.05, -47.11], [9E9, 9E9, 9E9, 9E9, 9E9, 9E9]];
	VAR jointtarget CDP_2193 := [[-13.5, 37.17, 3.72, 0, 49.11, -60.35], [9E9, 9E9, 9E9, 9E9, 9E9, 9E9]];
	VAR jointtarget CDP_2194 := [[-13.34, 37.22, 3.63, 0, 49.15, -73.59], [9E9, 9E9, 9E9, 9E9, 9E9, 9E9]];
	VAR jointtarget CDP_2195 := [[-13.18, 37.23, 3.61, 0, 49.16, -86.81], [9E9, 9E9, 9E9, 9E9, 9E9, 9E9]];
	VAR jointtarget CDP_2196 := [[-13.02, 37.2, 3.67, 0, 49.13, -100.04], [9E9, 9E9, 9E9, 9E9, 9E9, 9E9]];
	VAR jointtarget CDP_2197 := [[-12.88, 37.13, 3.79, 0, 49.08, -113.28], [9E9, 9E9, 9E9, 9E9, 9E9, 9E9]];
	VAR jointtarget CDP_2198 := [[-12.75, 37.02, 3.97, 0, 49, -126.54], [9E9, 9E9, 9E9, 9E9, 9E9, 9E9]];
	VAR jointtarget CDP_2199 := [[-12.64, 36.88, 4.21, 0, 48.9, -139.82], [9E9, 9E9, 9E9, 9E9, 9E9, 9E9]];
	VAR jointtarget CDP_2200 := [[-12.62, 36.84, 4.28, 0, 48.87, -146.49], [9E9, 9E9, 9E9, 9E9, 9E9, 9E9]];
	VAR jointtarget CDP_2201 := [[-12.59, 36.8, 4.35, 0, 48.85, -146.47], [9E9, 9E9, 9E9, 9E9, 9E9, 9E9]];
	VAR jointtarget CDP_2202 := [[-12.57, 36.76, 4.42, 0, 48.82, -146.44], [9E9, 9E9, 9E9, 9E9, 9E9, 9E9]];
	VAR jointtarget CDP_2203 := [[-12.54, 36.72, 4.49, 0, 48.79, -146.42], [9E9, 9E9, 9E9, 9E9, 9E9, 9E9]];
	VAR jointtarget CDP_2204 := [[-12.52, 36.68, 4.57, 0, 48.76, -146.4], [9E9, 9E9, 9E9, 9E9, 9E9, 9E9]];
	VAR jointtarget CDP_2205 := [[-12.49, 36.64, 4.64, 0, 48.73, -146.37], [9E9, 9E9, 9E9, 9E9, 9E9, 9E9]];
	VAR jointtarget CDP_2206 := [[-12.47, 36.6, 4.71, 0, 48.7, -146.35], [9E9, 9E9, 9E9, 9E9, 9E9, 9E9]];
	VAR jointtarget CDP_2207 := [[-12.44, 36.56, 4.78, 0, 48.67, -146.32], [9E9, 9E9, 9E9, 9E9, 9E9, 9E9]];
	VAR jointtarget CDP_2208 := [[-12.42, 36.51, 4.85, 0, 48.64, -146.3], [9E9, 9E9, 9E9, 9E9, 9E9, 9E9]];
	VAR jointtarget CDP_2209 := [[-12.39, 36.47, 4.92, 0, 48.61, -146.27], [9E9, 9E9, 9E9, 9E9, 9E9, 9E9]];
	VAR jointtarget CDP_2210 := [[-12.37, 36.43, 4.99, 0, 48.58, -146.25], [9E9, 9E9, 9E9, 9E9, 9E9, 9E9]];
	VAR jointtarget CDP_2211 := [[-12.34, 36.39, 5.06, 0, 48.55, -146.22], [9E9, 9E9, 9E9, 9E9, 9E9, 9E9]];
	VAR jointtarget CDP_2212 := [[-12.32, 36.35, 5.13, 0, 48.52, -146.2], [9E9, 9E9, 9E9, 9E9, 9E9, 9E9]];
	VAR jointtarget CDP_2213 := [[-12.29, 36.31, 5.2, 0, 48.49, -146.17], [9E9, 9E9, 9E9, 9E9, 9E9, 9E9]];
	VAR jointtarget CDP_2214 := [[-12.27, 36.27, 5.27, 0, 48.46, -146.15], [9E9, 9E9, 9E9, 9E9, 9E9, 9E9]];
	VAR jointtarget CDP_2215 := [[-12.24, 36.23, 5.34, 0, 48.43, -146.12], [9E9, 9E9, 9E9, 9E9, 9E9, 9E9]];
	VAR jointtarget CDP_2216 := [[-12.22, 36.19, 5.41, 0, 48.4, -146.1], [9E9, 9E9, 9E9, 9E9, 9E9, 9E9]];
	VAR jointtarget CDP_2217 := [[-12.19, 36.15, 5.48, 0, 48.37, -146.07], [9E9, 9E9, 9E9, 9E9, 9E9, 9E9]];
	VAR jointtarget CDP_2218 := [[-12.17, 36.11, 5.55, 0, 48.34, -146.05], [9E9, 9E9, 9E9, 9E9, 9E9, 9E9]];
	VAR jointtarget CDP_2219 := [[-12.14, 36.06, 5.62, 0, 48.32, -146.02], [9E9, 9E9, 9E9, 9E9, 9E9, 9E9]];
	VAR jointtarget CDP_2220 := [[-12.14, 36.05, 5.64, 0, 48.31, -145.46], [9E9, 9E9, 9E9, 9E9, 9E9, 9E9]];
	VAR jointtarget CDP_2221 := [[-12.13, 36.04, 5.66, 0, 48.3, -144.35], [9E9, 9E9, 9E9, 9E9, 9E9, 9E9]];
	VAR jointtarget CDP_2222 := [[-12.12, 36.03, 5.68, 0, 48.29, -143.24], [9E9, 9E9, 9E9, 9E9, 9E9, 9E9]];
	VAR jointtarget CDP_2223 := [[-12.11, 36.01, 5.7, 0, 48.28, -142.13], [9E9, 9E9, 9E9, 9E9, 9E9, 9E9]];
	VAR jointtarget CDP_2224 := [[-12.1, 36, 5.72, 0, 48.27, -141.01], [9E9, 9E9, 9E9, 9E9, 9E9, 9E9]];
	VAR jointtarget CDP_2225 := [[-12.09, 35.99, 5.74, 0, 48.26, -139.9], [9E9, 9E9, 9E9, 9E9, 9E9, 9E9]];
	VAR jointtarget CDP_2226 := [[-12.08, 35.98, 5.76, 0, 48.26, -138.79], [9E9, 9E9, 9E9, 9E9, 9E9, 9E9]];
	VAR jointtarget CDP_2227 := [[-12.07, 35.97, 5.78, 0, 48.25, -137.68], [9E9, 9E9, 9E9, 9E9, 9E9, 9E9]];
	VAR jointtarget CDP_2228 := [[-12.06, 35.96, 5.8, 0, 48.24, -136.56], [9E9, 9E9, 9E9, 9E9, 9E9, 9E9]];
	VAR jointtarget CDP_2229 := [[-12.05, 35.95, 5.82, 0, 48.23, -135.45], [9E9, 9E9, 9E9, 9E9, 9E9, 9E9]];
	VAR jointtarget CDP_2230 := [[-12.04, 35.93, 5.84, 0, 48.23, -134.34], [9E9, 9E9, 9E9, 9E9, 9E9, 9E9]];
	VAR jointtarget CDP_2231 := [[-12.03, 35.92, 5.86, 0, 48.22, -133.22], [9E9, 9E9, 9E9, 9E9, 9E9, 9E9]];
	VAR jointtarget CDP_2232 := [[-12.02, 35.91, 5.87, 0, 48.21, -132.11], [9E9, 9E9, 9E9, 9E9, 9E9, 9E9]];
	VAR jointtarget CDP_2233 := [[-12.01, 35.9, 5.89, 0, 48.21, -130.99], [9E9, 9E9, 9E9, 9E9, 9E9, 9E9]];
	VAR jointtarget CDP_2234 := [[-12, 35.89, 5.91, 0, 48.2, -129.88], [9E9, 9E9, 9E9, 9E9, 9E9, 9E9]];
	VAR jointtarget CDP_2235 := [[-11.99, 35.88, 5.92, 0, 48.19, -128.76], [9E9, 9E9, 9E9, 9E9, 9E9, 9E9]];
	VAR jointtarget CDP_2236 := [[-11.98, 35.87, 5.94, 0, 48.19, -127.65], [9E9, 9E9, 9E9, 9E9, 9E9, 9E9]];
	VAR jointtarget CDP_2237 := [[-11.97, 35.86, 5.96, 0, 48.18, -126.53], [9E9, 9E9, 9E9, 9E9, 9E9, 9E9]];
	VAR jointtarget CDP_2238 := [[-11.96, 35.85, 5.97, 0, 48.17, -125.42], [9E9, 9E9, 9E9, 9E9, 9E9, 9E9]];
	VAR jointtarget CDP_2239 := [[-11.95, 35.85, 5.99, 0, 48.17, -124.3], [9E9, 9E9, 9E9, 9E9, 9E9, 9E9]];
	VAR jointtarget CDP_2240 := [[-11.94, 35.84, 6, 0, 48.16, -123.74], [9E9, 9E9, 9E9, 9E9, 9E9, 9E9]];
	VAR jointtarget CDP_2241 := [[-11.93, 35.83, 6.01, 0, 48.16, -123.73], [9E9, 9E9, 9E9, 9E9, 9E9, 9E9]];
	VAR jointtarget CDP_2242 := [[-11.92, 35.82, 6.02, 0, 48.15, -123.72], [9E9, 9E9, 9E9, 9E9, 9E9, 9E9]];
	VAR jointtarget CDP_2243 := [[-11.9, 35.81, 6.04, 0, 48.15, -123.71], [9E9, 9E9, 9E9, 9E9, 9E9, 9E9]];
	VAR jointtarget CDP_2244 := [[-11.89, 35.81, 6.05, 0, 48.14, -123.7], [9E9, 9E9, 9E9, 9E9, 9E9, 9E9]];
	VAR jointtarget CDP_2245 := [[-11.88, 35.8, 6.06, 0, 48.14, -123.69], [9E9, 9E9, 9E9, 9E9, 9E9, 9E9]];
	VAR jointtarget CDP_2246 := [[-11.87, 35.79, 6.07, 0, 48.13, -123.68], [9E9, 9E9, 9E9, 9E9, 9E9, 9E9]];
	VAR jointtarget CDP_2247 := [[-11.86, 35.78, 6.09, 0, 48.13, -123.66], [9E9, 9E9, 9E9, 9E9, 9E9, 9E9]];
	VAR jointtarget CDP_2248 := [[-11.85, 35.77, 6.1, 0, 48.13, -123.65], [9E9, 9E9, 9E9, 9E9, 9E9, 9E9]];
	VAR jointtarget CDP_2249 := [[-11.84, 35.77, 6.11, 0, 48.12, -123.64], [9E9, 9E9, 9E9, 9E9, 9E9, 9E9]];
	VAR jointtarget CDP_2250 := [[-11.83, 35.76, 6.13, 0, 48.12, -123.63], [9E9, 9E9, 9E9, 9E9, 9E9, 9E9]];
	VAR jointtarget CDP_2251 := [[-11.82, 35.75, 6.14, 0, 48.11, -123.62], [9E9, 9E9, 9E9, 9E9, 9E9, 9E9]];
	VAR jointtarget CDP_2252 := [[-11.81, 35.74, 6.15, 0, 48.11, -123.61], [9E9, 9E9, 9E9, 9E9, 9E9, 9E9]];
	VAR jointtarget CDP_2253 := [[-11.8, 35.74, 6.16, 0, 48.1, -123.6], [9E9, 9E9, 9E9, 9E9, 9E9, 9E9]];
	VAR jointtarget CDP_2254 := [[-11.79, 35.73, 6.18, 0, 48.1, -123.59], [9E9, 9E9, 9E9, 9E9, 9E9, 9E9]];
	VAR jointtarget CDP_2255 := [[-11.78, 35.72, 6.19, 0, 48.09, -123.58], [9E9, 9E9, 9E9, 9E9, 9E9, 9E9]];
	VAR jointtarget CDP_2256 := [[-11.77, 35.71, 6.2, 0, 48.09, -123.57], [9E9, 9E9, 9E9, 9E9, 9E9, 9E9]];
	VAR jointtarget CDP_2257 := [[-11.76, 35.7, 6.21, 0, 48.08, -123.56], [9E9, 9E9, 9E9, 9E9, 9E9, 9E9]];
	VAR jointtarget CDP_2258 := [[-11.75, 35.7, 6.23, 0, 48.08, -123.55], [9E9, 9E9, 9E9, 9E9, 9E9, 9E9]];
	VAR jointtarget CDP_2259 := [[-11.74, 35.69, 6.24, 0, 48.07, -123.54], [9E9, 9E9, 9E9, 9E9, 9E9, 9E9]];
	VAR jointtarget CDP_2260 := [[-10.65, 35.46, 6.64, 0, 47.91, -100.65], [9E9, 9E9, 9E9, 9E9, 9E9, 9E9]];
	VAR jointtarget CDP_2261 := [[-9.55, 35.25, 6.99, 0, 47.76, -99.55], [9E9, 9E9, 9E9, 9E9, 9E9, 9E9]];
	VAR jointtarget CDP_2262 := [[-8.44, 35.06, 7.31, 0, 47.63, -98.44], [9E9, 9E9, 9E9, 9E9, 9E9, 9E9]];
	VAR jointtarget CDP_2263 := [[-7.33, 34.9, 7.59, 0, 47.51, -97.33], [9E9, 9E9, 9E9, 9E9, 9E9, 9E9]];
	VAR jointtarget CDP_2264 := [[-6.21, 34.76, 7.83, 0, 47.41, -96.21], [9E9, 9E9, 9E9, 9E9, 9E9, 9E9]];
	VAR jointtarget CDP_2265 := [[-5.09, 34.64, 8.03, 0, 47.33, -95.09], [9E9, 9E9, 9E9, 9E9, 9E9, 9E9]];
	VAR jointtarget CDP_2266 := [[-3.96, 34.55, 8.19, 0, 47.27, -93.96], [9E9, 9E9, 9E9, 9E9, 9E9, 9E9]];
	VAR jointtarget CDP_2267 := [[-2.83, 34.48, 8.31, 0, 47.22, -92.83], [9E9, 9E9, 9E9, 9E9, 9E9, 9E9]];
	VAR jointtarget CDP_2268 := [[-1.7, 34.43, 8.39, 0, 47.19, -91.7], [9E9, 9E9, 9E9, 9E9, 9E9, 9E9]];
	VAR jointtarget CDP_2269 := [[-0.56, 34.41, 8.43, 0, 47.17, -90.56], [9E9, 9E9, 9E9, 9E9, 9E9, 9E9]];
	VAR jointtarget CDP_2270 := [[0.57, 34.41, 8.43, 0, 47.17, -89.43], [9E9, 9E9, 9E9, 9E9, 9E9, 9E9]];
	VAR jointtarget CDP_2271 := [[1.7, 34.43, 8.39, 0, 47.19, -88.3], [9E9, 9E9, 9E9, 9E9, 9E9, 9E9]];
	VAR jointtarget CDP_2272 := [[2.84, 34.48, 8.31, 0, 47.22, -87.16], [9E9, 9E9, 9E9, 9E9, 9E9, 9E9]];
	VAR jointtarget CDP_2273 := [[3.97, 34.55, 8.19, 0, 47.27, -86.03], [9E9, 9E9, 9E9, 9E9, 9E9, 9E9]];
	VAR jointtarget CDP_2274 := [[5.09, 34.64, 8.03, 0, 47.33, -84.91], [9E9, 9E9, 9E9, 9E9, 9E9, 9E9]];
	VAR jointtarget CDP_2275 := [[6.22, 34.76, 7.83, 0, 47.42, -83.78], [9E9, 9E9, 9E9, 9E9, 9E9, 9E9]];
	VAR jointtarget CDP_2276 := [[7.34, 34.9, 7.59, 0, 47.51, -82.66], [9E9, 9E9, 9E9, 9E9, 9E9, 9E9]];
	VAR jointtarget CDP_2277 := [[8.45, 35.06, 7.31, 0, 47.63, -81.55], [9E9, 9E9, 9E9, 9E9, 9E9, 9E9]];
	VAR jointtarget CDP_2278 := [[9.56, 35.25, 6.99, 0, 47.76, -80.44], [9E9, 9E9, 9E9, 9E9, 9E9, 9E9]];
	VAR jointtarget CDP_2279 := [[10.65, 35.46, 6.63, 0, 47.91, -79.35], [9E9, 9E9, 9E9, 9E9, 9E9, 9E9]];
	VAR jointtarget CDP_2280 := [[10.71, 35.47, 6.61, 0, 47.92, -78.19], [9E9, 9E9, 9E9, 9E9, 9E9, 9E9]];
	VAR jointtarget CDP_2281 := [[10.76, 35.48, 6.59, 0, 47.93, -75.95], [9E9, 9E9, 9E9, 9E9, 9E9, 9E9]];
	VAR jointtarget CDP_2282 := [[10.82, 35.5, 6.56, 0, 47.94, -73.7], [9E9, 9E9, 9E9, 9E9, 9E9, 9E9]];
	VAR jointtarget CDP_2283 := [[10.87, 35.52, 6.53, 0, 47.95, -71.45], [9E9, 9E9, 9E9, 9E9, 9E9, 9E9]];
	VAR jointtarget CDP_2284 := [[10.92, 35.54, 6.49, 0, 47.97, -69.2], [9E9, 9E9, 9E9, 9E9, 9E9, 9E9]];
	VAR jointtarget CDP_2285 := [[10.97, 35.57, 6.45, 0, 47.99, -66.96], [9E9, 9E9, 9E9, 9E9, 9E9, 9E9]];
	VAR jointtarget CDP_2286 := [[11.03, 35.59, 6.41, 0, 48, -64.72], [9E9, 9E9, 9E9, 9E9, 9E9, 9E9]];
	VAR jointtarget CDP_2287 := [[11.07, 35.62, 6.36, 0, 48.02, -62.47], [9E9, 9E9, 9E9, 9E9, 9E9, 9E9]];
	VAR jointtarget CDP_2288 := [[11.12, 35.65, 6.31, 0, 48.04, -60.23], [9E9, 9E9, 9E9, 9E9, 9E9, 9E9]];
	VAR jointtarget CDP_2289 := [[11.17, 35.68, 6.25, 0, 48.07, -57.99], [9E9, 9E9, 9E9, 9E9, 9E9, 9E9]];
	VAR jointtarget CDP_2290 := [[11.22, 35.71, 6.2, 0, 48.09, -55.75], [9E9, 9E9, 9E9, 9E9, 9E9, 9E9]];
	VAR jointtarget CDP_2291 := [[11.26, 35.75, 6.13, 0, 48.12, -53.51], [9E9, 9E9, 9E9, 9E9, 9E9, 9E9]];
	VAR jointtarget CDP_2292 := [[11.3, 35.79, 6.07, 0, 48.14, -51.27], [9E9, 9E9, 9E9, 9E9, 9E9, 9E9]];
	VAR jointtarget CDP_2293 := [[11.35, 35.83, 6, 0, 48.17, -49.04], [9E9, 9E9, 9E9, 9E9, 9E9, 9E9]];
	VAR jointtarget CDP_2294 := [[11.39, 35.87, 5.93, 0, 48.2, -46.8], [9E9, 9E9, 9E9, 9E9, 9E9, 9E9]];
	VAR jointtarget CDP_2295 := [[11.43, 35.91, 5.86, 0, 48.23, -44.57], [9E9, 9E9, 9E9, 9E9, 9E9, 9E9]];
	VAR jointtarget CDP_2296 := [[11.46, 35.96, 5.78, 0, 48.26, -42.34], [9E9, 9E9, 9E9, 9E9, 9E9, 9E9]];
	VAR jointtarget CDP_2297 := [[11.5, 36, 5.7, 0, 48.3, -40.11], [9E9, 9E9, 9E9, 9E9, 9E9, 9E9]];
	VAR jointtarget CDP_2298 := [[11.53, 36.05, 5.62, 0, 48.33, -37.88], [9E9, 9E9, 9E9, 9E9, 9E9, 9E9]];
	VAR jointtarget CDP_2299 := [[11.57, 36.1, 5.54, 0, 48.36, -35.65], [9E9, 9E9, 9E9, 9E9, 9E9, 9E9]];
	VAR jointtarget CDP_2300 := [[11.59, 36.13, 5.49, 0, 48.39, -34.54], [9E9, 9E9, 9E9, 9E9, 9E9, 9E9]];
	VAR jointtarget CDP_2301 := [[11.6, 36.16, 5.43, 0, 48.41, -34.52], [9E9, 9E9, 9E9, 9E9, 9E9, 9E9]];
	VAR jointtarget CDP_2302 := [[11.62, 36.19, 5.38, 0, 48.43, -34.5], [9E9, 9E9, 9E9, 9E9, 9E9, 9E9]];
	VAR jointtarget CDP_2303 := [[11.64, 36.22, 5.33, 0, 48.45, -34.48], [9E9, 9E9, 9E9, 9E9, 9E9, 9E9]];
	VAR jointtarget CDP_2304 := [[11.66, 36.25, 5.28, 0, 48.47, -34.46], [9E9, 9E9, 9E9, 9E9, 9E9, 9E9]];
	VAR jointtarget CDP_2305 := [[11.68, 36.28, 5.23, 0, 48.49, -34.44], [9E9, 9E9, 9E9, 9E9, 9E9, 9E9]];
	VAR jointtarget CDP_2306 := [[11.7, 36.31, 5.18, 0, 48.52, -34.42], [9E9, 9E9, 9E9, 9E9, 9E9, 9E9]];
	VAR jointtarget CDP_2307 := [[11.72, 36.34, 5.12, 0, 48.54, -34.41], [9E9, 9E9, 9E9, 9E9, 9E9, 9E9]];
	VAR jointtarget CDP_2308 := [[11.74, 36.37, 5.07, 0, 48.56, -34.39], [9E9, 9E9, 9E9, 9E9, 9E9, 9E9]];
	VAR jointtarget CDP_2309 := [[11.76, 36.4, 5.02, 0, 48.58, -34.37], [9E9, 9E9, 9E9, 9E9, 9E9, 9E9]];
	VAR jointtarget CDP_2310 := [[11.77, 36.43, 4.97, 0, 48.6, -34.35], [9E9, 9E9, 9E9, 9E9, 9E9, 9E9]];
	VAR jointtarget CDP_2311 := [[11.79, 36.46, 4.92, 0, 48.62, -34.33], [9E9, 9E9, 9E9, 9E9, 9E9, 9E9]];
	VAR jointtarget CDP_2312 := [[11.81, 36.49, 4.86, 0, 48.65, -34.31], [9E9, 9E9, 9E9, 9E9, 9E9, 9E9]];
	VAR jointtarget CDP_2313 := [[11.83, 36.52, 4.81, 0, 48.67, -34.29], [9E9, 9E9, 9E9, 9E9, 9E9, 9E9]];
	VAR jointtarget CDP_2314 := [[11.85, 36.55, 4.76, 0, 48.69, -34.27], [9E9, 9E9, 9E9, 9E9, 9E9, 9E9]];
	VAR jointtarget CDP_2315 := [[11.87, 36.58, 4.71, 0, 48.71, -34.26], [9E9, 9E9, 9E9, 9E9, 9E9, 9E9]];
	VAR jointtarget CDP_2316 := [[11.89, 36.61, 4.66, 0, 48.73, -34.24], [9E9, 9E9, 9E9, 9E9, 9E9, 9E9]];
	VAR jointtarget CDP_2317 := [[11.91, 36.64, 4.6, 0, 48.75, -34.22], [9E9, 9E9, 9E9, 9E9, 9E9, 9E9]];
	VAR jointtarget CDP_2318 := [[11.92, 36.67, 4.55, 0, 48.78, -34.2], [9E9, 9E9, 9E9, 9E9, 9E9, 9E9]];
	VAR jointtarget CDP_2319 := [[11.94, 36.7, 4.5, 0, 48.8, -34.18], [9E9, 9E9, 9E9, 9E9, 9E9, 9E9]];
	VAR jointtarget CDP_2320 := [[12.05, 36.84, 4.27, 0, 48.9, -40.77], [9E9, 9E9, 9E9, 9E9, 9E9, 9E9]];
	VAR jointtarget CDP_2321 := [[12.18, 36.94, 4.08, 0, 48.97, -54.03], [9E9, 9E9, 9E9, 9E9, 9E9, 9E9]];
	VAR jointtarget CDP_2322 := [[12.33, 37.01, 3.96, 0, 49.02, -67.26], [9E9, 9E9, 9E9, 9E9, 9E9, 9E9]];
	VAR jointtarget CDP_2323 := [[12.49, 37.04, 3.91, 0, 49.04, -80.49], [9E9, 9E9, 9E9, 9E9, 9E9, 9E9]];
	VAR jointtarget CDP_2324 := [[12.65, 37.03, 3.93, 0, 49.04, -93.72], [9E9, 9E9, 9E9, 9E9, 9E9, 9E9]];
	VAR jointtarget CDP_2325 := [[12.8, 36.98, 4.03, 0, 49, -106.95], [9E9, 9E9, 9E9, 9E9, 9E9, 9E9]];
	VAR jointtarget CDP_2326 := [[12.94, 36.89, 4.18, 0, 48.93, -120.2], [9E9, 9E9, 9E9, 9E9, 9E9, 9E9]];
	VAR jointtarget CDP_2327 := [[13.06, 36.76, 4.39, 0, 48.84, -133.47], [9E9, 9E9, 9E9, 9E9, 9E9, 9E9]];
	VAR jointtarget CDP_2328 := [[13.15, 36.61, 4.65, 0, 48.73, -146.77], [9E9, 9E9, 9E9, 9E9, 9E9, 9E9]];
	VAR jointtarget CDP_2329 := [[13.2, 36.44, 4.94, 0, 48.61, -160.1], [9E9, 9E9, 9E9, 9E9, 9E9, 9E9]];
	VAR jointtarget CDP_2330 := [[13.22, 36.27, 5.25, 0, 48.49, -173.47], [9E9, 9E9, 9E9, 9E9, 9E9, 9E9]];
	VAR jointtarget CDP_2331 := [[13.2, 36.09, 5.55, 0, 48.36, -186.88], [9E9, 9E9, 9E9, 9E9, 9E9, 9E9]];
	VAR jointtarget CDP_2332 := [[13.15, 35.92, 5.84, 0, 48.24, -200.32], [9E9, 9E9, 9E9, 9E9, 9E9, 9E9]];
	VAR jointtarget CDP_2333 := [[13.06, 35.77, 6.09, 0, 48.13, -213.8], [9E9, 9E9, 9E9, 9E9, 9E9, 9E9]];
	VAR jointtarget CDP_2334 := [[12.93, 35.65, 6.3, 0, 48.05, -227.31], [9E9, 9E9, 9E9, 9E9, 9E9, 9E9]];
	VAR jointtarget CDP_2335 := [[12.79, 35.57, 6.45, 0, 47.99, -240.84], [9E9, 9E9, 9E9, 9E9, 9E9, 9E9]];
	VAR jointtarget CDP_2336 := [[12.63, 35.52, 6.53, 0, 47.95, -254.39], [9E9, 9E9, 9E9, 9E9, 9E9, 9E9]];
	VAR jointtarget CDP_2337 := [[12.47, 35.51, 6.54, 0, 47.95, -267.94], [9E9, 9E9, 9E9, 9E9, 9E9, 9E9]];
	VAR jointtarget CDP_2338 := [[12.3, 35.55, 6.48, 0, 47.97, -281.49], [9E9, 9E9, 9E9, 9E9, 9E9, 9E9]];
	VAR jointtarget CDP_2339 := [[12.15, 35.62, 6.35, 0, 48.03, -295.03], [9E9, 9E9, 9E9, 9E9, 9E9, 9E9]];
	VAR jointtarget CDP_2340 := [[12.13, 35.64, 6.32, 0, 48.04, -301.75], [9E9, 9E9, 9E9, 9E9, 9E9, 9E9]];
	VAR jointtarget CDP_2341 := [[12.1, 35.66, 6.29, 0, 48.05, -301.78], [9E9, 9E9, 9E9, 9E9, 9E9, 9E9]];
	VAR jointtarget CDP_2342 := [[12.07, 35.68, 6.25, 0, 48.07, -301.81], [9E9, 9E9, 9E9, 9E9, 9E9, 9E9]];
	VAR jointtarget CDP_2343 := [[12.04, 35.7, 6.22, 0, 48.08, -301.84], [9E9, 9E9, 9E9, 9E9, 9E9, 9E9]];
	VAR jointtarget CDP_2344 := [[12.01, 35.72, 6.19, 0, 48.09, -301.87], [9E9, 9E9, 9E9, 9E9, 9E9, 9E9]];
	VAR jointtarget CDP_2345 := [[11.98, 35.74, 6.16, 0, 48.11, -301.89], [9E9, 9E9, 9E9, 9E9, 9E9, 9E9]];
	VAR jointtarget CDP_2346 := [[11.95, 35.76, 6.12, 0, 48.12, -301.92], [9E9, 9E9, 9E9, 9E9, 9E9, 9E9]];
	VAR jointtarget CDP_2347 := [[11.92, 35.78, 6.09, 0, 48.13, -301.95], [9E9, 9E9, 9E9, 9E9, 9E9, 9E9]];
	VAR jointtarget CDP_2348 := [[11.9, 35.8, 6.06, 0, 48.15, -301.98], [9E9, 9E9, 9E9, 9E9, 9E9, 9E9]];
	VAR jointtarget CDP_2349 := [[11.87, 35.81, 6.02, 0, 48.16, -302.01], [9E9, 9E9, 9E9, 9E9, 9E9, 9E9]];
	VAR jointtarget CDP_2350 := [[11.84, 35.83, 5.99, 0, 48.18, -302.04], [9E9, 9E9, 9E9, 9E9, 9E9, 9E9]];
	VAR jointtarget CDP_2351 := [[11.81, 35.85, 5.96, 0, 48.19, -302.07], [9E9, 9E9, 9E9, 9E9, 9E9, 9E9]];
	VAR jointtarget CDP_2352 := [[11.78, 35.87, 5.92, 0, 48.2, -302.09], [9E9, 9E9, 9E9, 9E9, 9E9, 9E9]];
	VAR jointtarget CDP_2353 := [[11.75, 35.89, 5.89, 0, 48.22, -302.12], [9E9, 9E9, 9E9, 9E9, 9E9, 9E9]];
	VAR jointtarget CDP_2354 := [[11.73, 35.91, 5.86, 0, 48.23, -302.15], [9E9, 9E9, 9E9, 9E9, 9E9, 9E9]];
	VAR jointtarget CDP_2355 := [[11.7, 35.93, 5.82, 0, 48.24, -302.18], [9E9, 9E9, 9E9, 9E9, 9E9, 9E9]];
	VAR jointtarget CDP_2356 := [[11.67, 35.95, 5.79, 0, 48.26, -302.21], [9E9, 9E9, 9E9, 9E9, 9E9, 9E9]];
	VAR jointtarget CDP_2357 := [[11.64, 35.97, 5.76, 0, 48.27, -302.24], [9E9, 9E9, 9E9, 9E9, 9E9, 9E9]];
	VAR jointtarget CDP_2358 := [[11.61, 35.99, 5.72, 0, 48.29, -302.27], [9E9, 9E9, 9E9, 9E9, 9E9, 9E9]];
	VAR jointtarget CDP_2359 := [[11.58, 36.01, 5.69, 0, 48.3, -302.29], [9E9, 9E9, 9E9, 9E9, 9E9, 9E9]];
	VAR jointtarget CDP_2360 := [[11.54, 36.04, 5.64, 0, 48.32, -301.24], [9E9, 9E9, 9E9, 9E9, 9E9, 9E9]];
	VAR jointtarget CDP_2361 := [[11.49, 36.07, 5.59, 0, 48.34, -299.1], [9E9, 9E9, 9E9, 9E9, 9E9, 9E9]];
	VAR jointtarget CDP_2362 := [[11.44, 36.1, 5.54, 0, 48.36, -296.95], [9E9, 9E9, 9E9, 9E9, 9E9, 9E9]];
	VAR jointtarget CDP_2363 := [[11.39, 36.12, 5.5, 0, 48.38, -294.81], [9E9, 9E9, 9E9, 9E9, 9E9, 9E9]];
	VAR jointtarget CDP_2364 := [[11.34, 36.14, 5.46, 0, 48.4, -292.67], [9E9, 9E9, 9E9, 9E9, 9E9, 9E9]];
	VAR jointtarget CDP_2365 := [[11.28, 36.17, 5.42, 0, 48.41, -290.53], [9E9, 9E9, 9E9, 9E9, 9E9, 9E9]];
	VAR jointtarget CDP_2366 := [[11.23, 36.18, 5.39, 0, 48.43, -288.38], [9E9, 9E9, 9E9, 9E9, 9E9, 9E9]];
	VAR jointtarget CDP_2367 := [[11.18, 36.2, 5.36, 0, 48.44, -286.24], [9E9, 9E9, 9E9, 9E9, 9E9, 9E9]];
	VAR jointtarget CDP_2368 := [[11.13, 36.22, 5.33, 0, 48.45, -284.1], [9E9, 9E9, 9E9, 9E9, 9E9, 9E9]];
	VAR jointtarget CDP_2369 := [[11.07, 36.23, 5.31, 0, 48.46, -281.96], [9E9, 9E9, 9E9, 9E9, 9E9, 9E9]];
	VAR jointtarget CDP_2370 := [[11.02, 36.24, 5.3, 0, 48.47, -279.82], [9E9, 9E9, 9E9, 9E9, 9E9, 9E9]];
	VAR jointtarget CDP_2371 := [[10.96, 36.25, 5.28, 0, 48.47, -277.69], [9E9, 9E9, 9E9, 9E9, 9E9, 9E9]];
	VAR jointtarget CDP_2372 := [[10.91, 36.25, 5.27, 0, 48.48, -275.55], [9E9, 9E9, 9E9, 9E9, 9E9, 9E9]];
	VAR jointtarget CDP_2373 := [[10.85, 36.26, 5.27, 0, 48.48, -273.41], [9E9, 9E9, 9E9, 9E9, 9E9, 9E9]];
	VAR jointtarget CDP_2374 := [[10.8, 36.26, 5.26, 0, 48.48, -271.27], [9E9, 9E9, 9E9, 9E9, 9E9, 9E9]];
	VAR jointtarget CDP_2375 := [[10.74, 36.26, 5.26, 0, 48.48, -269.13], [9E9, 9E9, 9E9, 9E9, 9E9, 9E9]];
	VAR jointtarget CDP_2376 := [[10.69, 36.25, 5.27, 0, 48.48, -266.99], [9E9, 9E9, 9E9, 9E9, 9E9, 9E9]];
	VAR jointtarget CDP_2377 := [[10.63, 36.25, 5.28, 0, 48.47, -264.85], [9E9, 9E9, 9E9, 9E9, 9E9, 9E9]];
	VAR jointtarget CDP_2378 := [[10.58, 36.24, 5.29, 0, 48.47, -262.71], [9E9, 9E9, 9E9, 9E9, 9E9, 9E9]];
	VAR jointtarget CDP_2379 := [[10.52, 36.23, 5.31, 0, 48.46, -260.58], [9E9, 9E9, 9E9, 9E9, 9E9, 9E9]];
	VAR jointtarget CDP_2380 := [[9.44, 36.02, 5.66, 0, 48.31, -260.56], [9E9, 9E9, 9E9, 9E9, 9E9, 9E9]];
	VAR jointtarget CDP_2381 := [[8.36, 35.84, 5.98, 0, 48.18, -261.64], [9E9, 9E9, 9E9, 9E9, 9E9, 9E9]];
	VAR jointtarget CDP_2382 := [[7.27, 35.68, 6.26, 0, 48.07, -262.73], [9E9, 9E9, 9E9, 9E9, 9E9, 9E9]];
	VAR jointtarget CDP_2383 := [[6.17, 35.54, 6.49, 0, 47.97, -263.83], [9E9, 9E9, 9E9, 9E9, 9E9, 9E9]];
	VAR jointtarget CDP_2384 := [[5.07, 35.42, 6.69, 0, 47.88, -264.93], [9E9, 9E9, 9E9, 9E9, 9E9, 9E9]];
	VAR jointtarget CDP_2385 := [[3.97, 35.33, 6.85, 0, 47.82, -266.03], [9E9, 9E9, 9E9, 9E9, 9E9, 9E9]];
	VAR jointtarget CDP_2386 := [[2.86, 35.26, 6.97, 0, 47.77, -267.14], [9E9, 9E9, 9E9, 9E9, 9E9, 9E9]];
	VAR jointtarget CDP_2387 := [[1.75, 35.21, 7.05, 0, 47.73, -268.25], [9E9, 9E9, 9E9, 9E9, 9E9, 9E9]];
	VAR jointtarget CDP_2388 := [[0.64, 35.19, 7.1, 0, 47.72, -269.36], [9E9, 9E9, 9E9, 9E9, 9E9, 9E9]];
	VAR jointtarget CDP_2389 := [[-0.47, 35.18, 7.1, 0, 47.72, -270.47], [9E9, 9E9, 9E9, 9E9, 9E9, 9E9]];
	VAR jointtarget CDP_2390 := [[-1.58, 35.21, 7.06, 0, 47.73, -271.58], [9E9, 9E9, 9E9, 9E9, 9E9, 9E9]];
	VAR jointtarget CDP_2391 := [[-2.69, 35.25, 6.99, 0, 47.76, -272.69], [9E9, 9E9, 9E9, 9E9, 9E9, 9E9]];
	VAR jointtarget CDP_2392 := [[-3.8, 35.32, 6.87, 0, 47.81, -273.8], [9E9, 9E9, 9E9, 9E9, 9E9, 9E9]];
	VAR jointtarget CDP_2393 := [[-4.9, 35.41, 6.72, 0, 47.87, -274.9], [9E9, 9E9, 9E9, 9E9, 9E9, 9E9]];
	VAR jointtarget CDP_2394 := [[-6, 35.52, 6.53, 0, 47.95, -276], [9E9, 9E9, 9E9, 9E9, 9E9, 9E9]];
	VAR jointtarget CDP_2395 := [[-7.1, 35.66, 6.3, 0, 48.05, -277.1], [9E9, 9E9, 9E9, 9E9, 9E9, 9E9]];
	VAR jointtarget CDP_2396 := [[-8.19, 35.81, 6.02, 0, 48.16, -278.19], [9E9, 9E9, 9E9, 9E9, 9E9, 9E9]];
	VAR jointtarget CDP_2397 := [[-9.28, 35.99, 5.72, 0, 48.29, -279.28], [9E9, 9E9, 9E9, 9E9, 9E9, 9E9]];
	VAR jointtarget CDP_2398 := [[-10.36, 36.2, 5.37, 0, 48.44, -280.36], [9E9, 9E9, 9E9, 9E9, 9E9, 9E9]];
	VAR jointtarget CDP_2399 := [[-11.43, 36.42, 4.98, 0, 48.6, -281.43], [9E9, 9E9, 9E9, 9E9, 9E9, 9E9]];
	VAR jointtarget CDP_2400 := [[-11.44, 36.43, 4.97, 0, 48.6, -281.78], [9E9, 9E9, 9E9, 9E9, 9E9, 9E9]];
	VAR jointtarget CDP_2401 := [[-11.46, 36.43, 4.97, 0, 48.6, -282.45], [9E9, 9E9, 9E9, 9E9, 9E9, 9E9]];
	VAR jointtarget CDP_2402 := [[-11.48, 36.44, 4.96, 0, 48.61, -283.13], [9E9, 9E9, 9E9, 9E9, 9E9, 9E9]];
	VAR jointtarget CDP_2403 := [[-11.49, 36.44, 4.95, 0, 48.61, -283.81], [9E9, 9E9, 9E9, 9E9, 9E9, 9E9]];
	VAR jointtarget CDP_2404 := [[-11.51, 36.44, 4.94, 0, 48.61, -284.49], [9E9, 9E9, 9E9, 9E9, 9E9, 9E9]];
	VAR jointtarget CDP_2405 := [[-11.53, 36.45, 4.93, 0, 48.62, -285.17], [9E9, 9E9, 9E9, 9E9, 9E9, 9E9]];
	VAR jointtarget CDP_2406 := [[-11.54, 36.45, 4.93, 0, 48.62, -285.84], [9E9, 9E9, 9E9, 9E9, 9E9, 9E9]];
	VAR jointtarget CDP_2407 := [[-11.56, 36.46, 4.92, 0, 48.62, -286.52], [9E9, 9E9, 9E9, 9E9, 9E9, 9E9]];
	VAR jointtarget CDP_2408 := [[-11.57, 36.46, 4.91, 0, 48.63, -287.2], [9E9, 9E9, 9E9, 9E9, 9E9, 9E9]];
	VAR jointtarget CDP_2409 := [[-11.59, 36.47, 4.9, 0, 48.63, -287.88], [9E9, 9E9, 9E9, 9E9, 9E9, 9E9]];
	VAR jointtarget CDP_2410 := [[-11.6, 36.48, 4.89, 0, 48.64, -288.56], [9E9, 9E9, 9E9, 9E9, 9E9, 9E9]];
	VAR jointtarget CDP_2411 := [[-11.62, 36.48, 4.88, 0, 48.64, -289.23], [9E9, 9E9, 9E9, 9E9, 9E9, 9E9]];
	VAR jointtarget CDP_2412 := [[-11.64, 36.49, 4.87, 0, 48.64, -289.91], [9E9, 9E9, 9E9, 9E9, 9E9, 9E9]];
	VAR jointtarget CDP_2413 := [[-11.65, 36.49, 4.86, 0, 48.65, -290.59], [9E9, 9E9, 9E9, 9E9, 9E9, 9E9]];
	VAR jointtarget CDP_2414 := [[-11.67, 36.5, 4.84, 0, 48.65, -291.27], [9E9, 9E9, 9E9, 9E9, 9E9, 9E9]];
	VAR jointtarget CDP_2415 := [[-11.68, 36.51, 4.83, 0, 48.66, -291.94], [9E9, 9E9, 9E9, 9E9, 9E9, 9E9]];
	VAR jointtarget CDP_2416 := [[-11.7, 36.52, 4.82, 0, 48.66, -292.62], [9E9, 9E9, 9E9, 9E9, 9E9, 9E9]];
	VAR jointtarget CDP_2417 := [[-11.71, 36.52, 4.81, 0, 48.67, -293.3], [9E9, 9E9, 9E9, 9E9, 9E9, 9E9]];
	VAR jointtarget CDP_2418 := [[-11.73, 36.53, 4.8, 0, 48.67, -293.98], [9E9, 9E9, 9E9, 9E9, 9E9, 9E9]];
	VAR jointtarget CDP_2419 := [[-11.74, 36.54, 4.78, 0, 48.68, -294.65], [9E9, 9E9, 9E9, 9E9, 9E9, 9E9]];
	VAR jointtarget CDP_2420 := [[-11.8, 36.57, 4.73, 0, 48.7, -295.04], [9E9, 9E9, 9E9, 9E9, 9E9, 9E9]];
	VAR jointtarget CDP_2421 := [[-11.86, 36.6, 4.68, 0, 48.72, -295.11], [9E9, 9E9, 9E9, 9E9, 9E9, 9E9]];
	VAR jointtarget CDP_2422 := [[-11.93, 36.63, 4.62, 0, 48.75, -295.17], [9E9, 9E9, 9E9, 9E9, 9E9, 9E9]];
	VAR jointtarget CDP_2423 := [[-11.99, 36.66, 4.57, 0, 48.77, -295.23], [9E9, 9E9, 9E9, 9E9, 9E9, 9E9]];
	VAR jointtarget CDP_2424 := [[-12.05, 36.69, 4.51, 0, 48.79, -295.29], [9E9, 9E9, 9E9, 9E9, 9E9, 9E9]];
	VAR jointtarget CDP_2425 := [[-12.11, 36.73, 4.46, 0, 48.82, -295.35], [9E9, 9E9, 9E9, 9E9, 9E9, 9E9]];
	VAR jointtarget CDP_2426 := [[-12.17, 36.76, 4.4, 0, 48.84, -295.41], [9E9, 9E9, 9E9, 9E9, 9E9, 9E9]];
	VAR jointtarget CDP_2427 := [[-12.23, 36.79, 4.35, 0, 48.86, -295.47], [9E9, 9E9, 9E9, 9E9, 9E9, 9E9]];
	VAR jointtarget CDP_2428 := [[-12.29, 36.82, 4.3, 0, 48.88, -295.53], [9E9, 9E9, 9E9, 9E9, 9E9, 9E9]];
	VAR jointtarget CDP_2429 := [[-12.35, 36.85, 4.24, 0, 48.91, -295.59], [9E9, 9E9, 9E9, 9E9, 9E9, 9E9]];
	VAR jointtarget CDP_2430 := [[-12.41, 36.89, 4.19, 0, 48.93, -295.65], [9E9, 9E9, 9E9, 9E9, 9E9, 9E9]];
	VAR jointtarget CDP_2431 := [[-12.47, 36.92, 4.13, 0, 48.95, -295.71], [9E9, 9E9, 9E9, 9E9, 9E9, 9E9]];
	VAR jointtarget CDP_2432 := [[-12.53, 36.95, 4.07, 0, 48.98, -295.77], [9E9, 9E9, 9E9, 9E9, 9E9, 9E9]];
	VAR jointtarget CDP_2433 := [[-12.59, 36.98, 4.02, 0, 49, -295.83], [9E9, 9E9, 9E9, 9E9, 9E9, 9E9]];
	VAR jointtarget CDP_2434 := [[-12.65, 37.01, 3.96, 0, 49.02, -295.89], [9E9, 9E9, 9E9, 9E9, 9E9, 9E9]];
	VAR jointtarget CDP_2435 := [[-12.71, 37.05, 3.91, 0, 49.05, -295.95], [9E9, 9E9, 9E9, 9E9, 9E9, 9E9]];
	VAR jointtarget CDP_2436 := [[-12.77, 37.08, 3.85, 0, 49.07, -296.01], [9E9, 9E9, 9E9, 9E9, 9E9, 9E9]];
	VAR jointtarget CDP_2437 := [[-12.83, 37.11, 3.8, 0, 49.09, -296.07], [9E9, 9E9, 9E9, 9E9, 9E9, 9E9]];
	VAR jointtarget CDP_2438 := [[-12.89, 37.14, 3.74, 0, 49.12, -296.13], [9E9, 9E9, 9E9, 9E9, 9E9, 9E9]];
	VAR jointtarget CDP_2439 := [[-12.95, 37.18, 3.68, 0, 49.14, -296.19], [9E9, 9E9, 9E9, 9E9, 9E9, 9E9]];
	VAR jointtarget CDP_2440 := [[-13.07, 37.23, 3.59, 0, 49.18, -291.14], [9E9, 9E9, 9E9, 9E9, 9E9, 9E9]];
	VAR jointtarget CDP_2441 := [[-13.19, 37.26, 3.55, 0, 49.2, -280.95], [9E9, 9E9, 9E9, 9E9, 9E9, 9E9]];
	VAR jointtarget CDP_2442 := [[-13.32, 37.26, 3.54, 0, 49.2, -270.75], [9E9, 9E9, 9E9, 9E9, 9E9, 9E9]];
	VAR jointtarget CDP_2443 := [[-13.45, 37.23, 3.58, 0, 49.18, -260.55], [9E9, 9E9, 9E9, 9E9, 9E9, 9E9]];
	VAR jointtarget CDP_2444 := [[-13.57, 37.18, 3.67, 0, 49.15, -250.35], [9E9, 9E9, 9E9, 9E9, 9E9, 9E9]];
	VAR jointtarget CDP_2445 := [[-13.68, 37.11, 3.79, 0, 49.09, -240.14], [9E9, 9E9, 9E9, 9E9, 9E9, 9E9]];
	VAR jointtarget CDP_2446 := [[-13.78, 37.02, 3.95, 0, 49.03, -229.91], [9E9, 9E9, 9E9, 9E9, 9E9, 9E9]];
	VAR jointtarget CDP_2447 := [[-13.86, 36.91, 4.14, 0, 48.95, -219.67], [9E9, 9E9, 9E9, 9E9, 9E9, 9E9]];
	VAR jointtarget CDP_2448 := [[-13.93, 36.78, 4.36, 0, 48.86, -209.41], [9E9, 9E9, 9E9, 9E9, 9E9, 9E9]];
	VAR jointtarget CDP_2449 := [[-13.97, 36.65, 4.59, 0, 48.76, -199.13], [9E9, 9E9, 9E9, 9E9, 9E9, 9E9]];
	VAR jointtarget CDP_2450 := [[-13.99, 36.51, 4.84, 0, 48.66, -188.83], [9E9, 9E9, 9E9, 9E9, 9E9, 9E9]];
	VAR jointtarget CDP_2451 := [[-13.98, 36.36, 5.08, 0, 48.55, -178.5], [9E9, 9E9, 9E9, 9E9, 9E9, 9E9]];
	VAR jointtarget CDP_2452 := [[-13.96, 36.22, 5.32, 0, 48.45, -168.15], [9E9, 9E9, 9E9, 9E9, 9E9, 9E9]];
	VAR jointtarget CDP_2453 := [[-13.91, 36.09, 5.55, 0, 48.36, -157.77], [9E9, 9E9, 9E9, 9E9, 9E9, 9E9]];
	VAR jointtarget CDP_2454 := [[-13.84, 35.97, 5.76, 0, 48.27, -147.38], [9E9, 9E9, 9E9, 9E9, 9E9, 9E9]];
	VAR jointtarget CDP_2455 := [[-13.75, 35.87, 5.93, 0, 48.2, -136.97], [9E9, 9E9, 9E9, 9E9, 9E9, 9E9]];
	VAR jointtarget CDP_2456 := [[-13.64, 35.78, 6.08, 0, 48.14, -126.54], [9E9, 9E9, 9E9, 9E9, 9E9, 9E9]];
	VAR jointtarget CDP_2457 := [[-13.52, 35.72, 6.19, 0, 48.09, -116.09], [9E9, 9E9, 9E9, 9E9, 9E9, 9E9]];
	VAR jointtarget CDP_2458 := [[-13.4, 35.68, 6.25, 0, 48.07, -105.64], [9E9, 9E9, 9E9, 9E9, 9E9, 9E9]];
	VAR jointtarget CDP_2459 := [[-13.27, 35.67, 6.28, 0, 48.06, -95.19], [9E9, 9E9, 9E9, 9E9, 9E9, 9E9]];
	VAR jointtarget CDP_2460 := [[-13.2, 35.67, 6.28, 0, 48.06, -89.96], [9E9, 9E9, 9E9, 9E9, 9E9, 9E9]];
	VAR jointtarget CDP_2461 := [[-13.13, 35.67, 6.28, 0, 48.06, -89.89], [9E9, 9E9, 9E9, 9E9, 9E9, 9E9]];
	VAR jointtarget CDP_2462 := [[-13.06, 35.67, 6.27, 0, 48.06, -89.82], [9E9, 9E9, 9E9, 9E9, 9E9, 9E9]];
	VAR jointtarget CDP_2463 := [[-12.99, 35.67, 6.27, 0, 48.06, -89.75], [9E9, 9E9, 9E9, 9E9, 9E9, 9E9]];
	VAR jointtarget CDP_2464 := [[-12.93, 35.66, 6.27, 0, 48.06, -89.69], [9E9, 9E9, 9E9, 9E9, 9E9, 9E9]];
	VAR jointtarget CDP_2465 := [[-12.86, 35.66, 6.27, 0, 48.06, -89.62], [9E9, 9E9, 9E9, 9E9, 9E9, 9E9]];
	VAR jointtarget CDP_2466 := [[-12.79, 35.66, 6.27, 0, 48.06, -89.55], [9E9, 9E9, 9E9, 9E9, 9E9, 9E9]];
	VAR jointtarget CDP_2467 := [[-12.72, 35.66, 6.27, 0, 48.06, -89.48], [9E9, 9E9, 9E9, 9E9, 9E9, 9E9]];
	VAR jointtarget CDP_2468 := [[-12.65, 35.66, 6.27, 0, 48.07, -89.41], [9E9, 9E9, 9E9, 9E9, 9E9, 9E9]];
	VAR jointtarget CDP_2469 := [[-12.59, 35.67, 6.27, 0, 48.07, -89.35], [9E9, 9E9, 9E9, 9E9, 9E9, 9E9]];
	VAR jointtarget CDP_2470 := [[-12.52, 35.67, 6.27, 0, 48.07, -89.28], [9E9, 9E9, 9E9, 9E9, 9E9, 9E9]];
	VAR jointtarget CDP_2471 := [[-12.45, 35.67, 6.26, 0, 48.07, -89.21], [9E9, 9E9, 9E9, 9E9, 9E9, 9E9]];
	VAR jointtarget CDP_2472 := [[-12.38, 35.67, 6.26, 0, 48.07, -89.14], [9E9, 9E9, 9E9, 9E9, 9E9, 9E9]];
	VAR jointtarget CDP_2473 := [[-12.32, 35.67, 6.26, 0, 48.07, -89.07], [9E9, 9E9, 9E9, 9E9, 9E9, 9E9]];
	VAR jointtarget CDP_2474 := [[-12.25, 35.67, 6.26, 0, 48.07, -89.01], [9E9, 9E9, 9E9, 9E9, 9E9, 9E9]];
	VAR jointtarget CDP_2475 := [[-12.18, 35.67, 6.26, 0, 48.08, -88.94], [9E9, 9E9, 9E9, 9E9, 9E9, 9E9]];
	VAR jointtarget CDP_2476 := [[-12.11, 35.67, 6.25, 0, 48.08, -88.87], [9E9, 9E9, 9E9, 9E9, 9E9, 9E9]];
	VAR jointtarget CDP_2477 := [[-12.04, 35.67, 6.25, 0, 48.08, -88.8], [9E9, 9E9, 9E9, 9E9, 9E9, 9E9]];
	VAR jointtarget CDP_2478 := [[-11.98, 35.67, 6.25, 0, 48.08, -88.74], [9E9, 9E9, 9E9, 9E9, 9E9, 9E9]];
	VAR jointtarget CDP_2479 := [[-11.91, 35.67, 6.24, 0, 48.08, -88.67], [9E9, 9E9, 9E9, 9E9, 9E9, 9E9]];
	VAR jointtarget CDP_2480 := [[-11.89, 35.67, 6.24, 0, 48.08, -88.98], [9E9, 9E9, 9E9, 9E9, 9E9, 9E9]];
	VAR jointtarget CDP_2481 := [[-11.87, 35.67, 6.24, 0, 48.08, -89.63], [9E9, 9E9, 9E9, 9E9, 9E9, 9E9]];
	VAR jointtarget CDP_2482 := [[-11.86, 35.67, 6.24, 0, 48.08, -90.27], [9E9, 9E9, 9E9, 9E9, 9E9, 9E9]];
	VAR jointtarget CDP_2483 := [[-11.84, 35.67, 6.24, 0, 48.08, -90.92], [9E9, 9E9, 9E9, 9E9, 9E9, 9E9]];
	VAR jointtarget CDP_2484 := [[-11.82, 35.67, 6.25, 0, 48.08, -91.56], [9E9, 9E9, 9E9, 9E9, 9E9, 9E9]];
	VAR jointtarget CDP_2485 := [[-11.81, 35.67, 6.25, 0, 48.08, -92.21], [9E9, 9E9, 9E9, 9E9, 9E9, 9E9]];
	VAR jointtarget CDP_2486 := [[-11.79, 35.67, 6.25, 0, 48.08, -92.85], [9E9, 9E9, 9E9, 9E9, 9E9, 9E9]];
	VAR jointtarget CDP_2487 := [[-11.77, 35.67, 6.25, 0, 48.08, -93.5], [9E9, 9E9, 9E9, 9E9, 9E9, 9E9]];
	VAR jointtarget CDP_2488 := [[-11.76, 35.67, 6.25, 0, 48.08, -94.14], [9E9, 9E9, 9E9, 9E9, 9E9, 9E9]];
	VAR jointtarget CDP_2489 := [[-11.74, 35.66, 6.26, 0, 48.08, -94.79], [9E9, 9E9, 9E9, 9E9, 9E9, 9E9]];
	VAR jointtarget CDP_2490 := [[-11.72, 35.66, 6.26, 0, 48.08, -95.43], [9E9, 9E9, 9E9, 9E9, 9E9, 9E9]];
	VAR jointtarget CDP_2491 := [[-11.71, 35.66, 6.26, 0, 48.08, -96.08], [9E9, 9E9, 9E9, 9E9, 9E9, 9E9]];
	VAR jointtarget CDP_2492 := [[-11.69, 35.66, 6.26, 0, 48.08, -96.72], [9E9, 9E9, 9E9, 9E9, 9E9, 9E9]];
	VAR jointtarget CDP_2493 := [[-11.67, 35.66, 6.27, 0, 48.07, -97.37], [9E9, 9E9, 9E9, 9E9, 9E9, 9E9]];
	VAR jointtarget CDP_2494 := [[-11.66, 35.65, 6.27, 0, 48.07, -98.01], [9E9, 9E9, 9E9, 9E9, 9E9, 9E9]];
	VAR jointtarget CDP_2495 := [[-11.64, 35.65, 6.28, 0, 48.07, -98.66], [9E9, 9E9, 9E9, 9E9, 9E9, 9E9]];
	VAR jointtarget CDP_2496 := [[-11.62, 35.65, 6.28, 0, 48.07, -99.31], [9E9, 9E9, 9E9, 9E9, 9E9, 9E9]];
	VAR jointtarget CDP_2497 := [[-11.61, 35.65, 6.29, 0, 48.07, -99.95], [9E9, 9E9, 9E9, 9E9, 9E9, 9E9]];
	VAR jointtarget CDP_2498 := [[-11.59, 35.64, 6.29, 0, 48.06, -100.6], [9E9, 9E9, 9E9, 9E9, 9E9, 9E9]];
	VAR jointtarget CDP_2499 := [[-11.57, 35.64, 6.3, 0, 48.06, -101.24], [9E9, 9E9, 9E9, 9E9, 9E9, 9E9]];
	VAR jointtarget CDP_2500 := [[-10.48, 35.41, 6.69, 0, 47.9, -100.48], [9E9, 9E9, 9E9, 9E9, 9E9, 9E9]];
	VAR jointtarget CDP_2501 := [[-9.38, 35.2, 7.04, 0, 47.75, -99.38], [9E9, 9E9, 9E9, 9E9, 9E9, 9E9]];
	VAR jointtarget CDP_2502 := [[-8.27, 35.02, 7.36, 0, 47.62, -98.27], [9E9, 9E9, 9E9, 9E9, 9E9, 9E9]];
	VAR jointtarget CDP_2503 := [[-7.15, 34.86, 7.63, 0, 47.51, -97.15], [9E9, 9E9, 9E9, 9E9, 9E9, 9E9]];
	VAR jointtarget CDP_2504 := [[-6.03, 34.72, 7.86, 0, 47.42, -96.03], [9E9, 9E9, 9E9, 9E9, 9E9, 9E9]];
	VAR jointtarget CDP_2505 := [[-4.9, 34.61, 8.05, 0, 47.34, -94.9], [9E9, 9E9, 9E9, 9E9, 9E9, 9E9]];
	VAR jointtarget CDP_2506 := [[-3.77, 34.52, 8.21, 0, 47.27, -93.77], [9E9, 9E9, 9E9, 9E9, 9E9, 9E9]];
	VAR jointtarget CDP_2507 := [[-2.64, 34.45, 8.32, 0, 47.23, -92.64], [9E9, 9E9, 9E9, 9E9, 9E9, 9E9]];
	VAR jointtarget CDP_2508 := [[-1.51, 34.41, 8.39, 0, 47.2, -91.51], [9E9, 9E9, 9E9, 9E9, 9E9, 9E9]];
	VAR jointtarget CDP_2509 := [[-0.37, 34.39, 8.43, 0, 47.18, -90.37], [9E9, 9E9, 9E9, 9E9, 9E9, 9E9]];
	VAR jointtarget CDP_2510 := [[0.76, 34.39, 8.42, 0, 47.19, -89.24], [9E9, 9E9, 9E9, 9E9, 9E9, 9E9]];
	VAR jointtarget CDP_2511 := [[1.9, 34.42, 8.37, 0, 47.21, -88.1], [9E9, 9E9, 9E9, 9E9, 9E9, 9E9]];
	VAR jointtarget CDP_2512 := [[3.03, 34.47, 8.29, 0, 47.24, -86.97], [9E9, 9E9, 9E9, 9E9, 9E9, 9E9]];
	VAR jointtarget CDP_2513 := [[4.16, 34.55, 8.16, 0, 47.29, -85.84], [9E9, 9E9, 9E9, 9E9, 9E9, 9E9]];
	VAR jointtarget CDP_2514 := [[5.29, 34.65, 7.99, 0, 47.36, -84.71], [9E9, 9E9, 9E9, 9E9, 9E9, 9E9]];
	VAR jointtarget CDP_2515 := [[6.42, 34.77, 7.79, 0, 47.45, -83.58], [9E9, 9E9, 9E9, 9E9, 9E9, 9E9]];
	VAR jointtarget CDP_2516 := [[7.54, 34.91, 7.54, 0, 47.55, -82.46], [9E9, 9E9, 9E9, 9E9, 9E9, 9E9]];
	VAR jointtarget CDP_2517 := [[8.65, 35.08, 7.25, 0, 47.67, -81.35], [9E9, 9E9, 9E9, 9E9, 9E9, 9E9]];
	VAR jointtarget CDP_2518 := [[9.76, 35.27, 6.93, 0, 47.8, -80.24], [9E9, 9E9, 9E9, 9E9, 9E9, 9E9]];
	VAR jointtarget CDP_2519 := [[10.86, 35.49, 6.56, 0, 47.95, -79.14], [9E9, 9E9, 9E9, 9E9, 9E9, 9E9]];
	VAR jointtarget CDP_2520 := [[10.87, 35.49, 6.56, 0, 47.96, -79.46], [9E9, 9E9, 9E9, 9E9, 9E9, 9E9]];
	VAR jointtarget CDP_2521 := [[10.89, 35.49, 6.55, 0, 47.96, -80.1], [9E9, 9E9, 9E9, 9E9, 9E9, 9E9]];
	VAR jointtarget CDP_2522 := [[10.91, 35.49, 6.55, 0, 47.96, -80.75], [9E9, 9E9, 9E9, 9E9, 9E9, 9E9]];
	VAR jointtarget CDP_2523 := [[10.92, 35.5, 6.54, 0, 47.96, -81.39], [9E9, 9E9, 9E9, 9E9, 9E9, 9E9]];
	VAR jointtarget CDP_2524 := [[10.94, 35.5, 6.54, 0, 47.96, -82.04], [9E9, 9E9, 9E9, 9E9, 9E9, 9E9]];
	VAR jointtarget CDP_2525 := [[10.96, 35.5, 6.53, 0, 47.97, -82.68], [9E9, 9E9, 9E9, 9E9, 9E9, 9E9]];
	VAR jointtarget CDP_2526 := [[10.97, 35.5, 6.53, 0, 47.97, -83.33], [9E9, 9E9, 9E9, 9E9, 9E9, 9E9]];
	VAR jointtarget CDP_2527 := [[10.99, 35.51, 6.53, 0, 47.97, -83.97], [9E9, 9E9, 9E9, 9E9, 9E9, 9E9]];
	VAR jointtarget CDP_2528 := [[11.01, 35.51, 6.52, 0, 47.97, -84.62], [9E9, 9E9, 9E9, 9E9, 9E9, 9E9]];
	VAR jointtarget CDP_2529 := [[11.02, 35.51, 6.52, 0, 47.97, -85.27], [9E9, 9E9, 9E9, 9E9, 9E9, 9E9]];
	VAR jointtarget CDP_2530 := [[11.04, 35.51, 6.52, 0, 47.97, -85.91], [9E9, 9E9, 9E9, 9E9, 9E9, 9E9]];
	VAR jointtarget CDP_2531 := [[11.06, 35.51, 6.52, 0, 47.97, -86.56], [9E9, 9E9, 9E9, 9E9, 9E9, 9E9]];
	VAR jointtarget CDP_2532 := [[11.07, 35.51, 6.51, 0, 47.97, -87.2], [9E9, 9E9, 9E9, 9E9, 9E9, 9E9]];
	VAR jointtarget CDP_2533 := [[11.09, 35.51, 6.51, 0, 47.97, -87.85], [9E9, 9E9, 9E9, 9E9, 9E9, 9E9]];
	VAR jointtarget CDP_2534 := [[11.11, 35.51, 6.51, 0, 47.97, -88.49], [9E9, 9E9, 9E9, 9E9, 9E9, 9E9]];
	VAR jointtarget CDP_2535 := [[11.13, 35.51, 6.51, 0, 47.97, -89.14], [9E9, 9E9, 9E9, 9E9, 9E9, 9E9]];
	VAR jointtarget CDP_2536 := [[11.14, 35.51, 6.51, 0, 47.97, -89.78], [9E9, 9E9, 9E9, 9E9, 9E9, 9E9]];
	VAR jointtarget CDP_2537 := [[11.16, 35.51, 6.51, 0, 47.97, -90.43], [9E9, 9E9, 9E9, 9E9, 9E9, 9E9]];
	VAR jointtarget CDP_2538 := [[11.18, 35.51, 6.51, 0, 47.97, -91.07], [9E9, 9E9, 9E9, 9E9, 9E9, 9E9]];
	VAR jointtarget CDP_2539 := [[11.19, 35.51, 6.51, 0, 47.97, -91.72], [9E9, 9E9, 9E9, 9E9, 9E9, 9E9]];
	VAR jointtarget CDP_2540 := [[11.26, 35.51, 6.52, 0, 47.97, -91.98], [9E9, 9E9, 9E9, 9E9, 9E9, 9E9]];
	VAR jointtarget CDP_2541 := [[11.33, 35.51, 6.52, 0, 47.97, -91.91], [9E9, 9E9, 9E9, 9E9, 9E9, 9E9]];
	VAR jointtarget CDP_2542 := [[11.4, 35.51, 6.53, 0, 47.97, -91.84], [9E9, 9E9, 9E9, 9E9, 9E9, 9E9]];
	VAR jointtarget CDP_2543 := [[11.47, 35.5, 6.53, 0, 47.97, -91.78], [9E9, 9E9, 9E9, 9E9, 9E9, 9E9]];
	VAR jointtarget CDP_2544 := [[11.53, 35.5, 6.53, 0, 47.96, -91.71], [9E9, 9E9, 9E9, 9E9, 9E9, 9E9]];
	VAR jointtarget CDP_2545 := [[11.6, 35.5, 6.54, 0, 47.96, -91.64], [9E9, 9E9, 9E9, 9E9, 9E9, 9E9]];
	VAR jointtarget CDP_2546 := [[11.67, 35.5, 6.54, 0, 47.96, -91.57], [9E9, 9E9, 9E9, 9E9, 9E9, 9E9]];
	VAR jointtarget CDP_2547 := [[11.74, 35.5, 6.54, 0, 47.96, -91.5], [9E9, 9E9, 9E9, 9E9, 9E9, 9E9]];
	VAR jointtarget CDP_2548 := [[11.81, 35.49, 6.55, 0, 47.96, -91.44], [9E9, 9E9, 9E9, 9E9, 9E9, 9E9]];
	VAR jointtarget CDP_2549 := [[11.87, 35.49, 6.55, 0, 47.96, -91.37], [9E9, 9E9, 9E9, 9E9, 9E9, 9E9]];
	VAR jointtarget CDP_2550 := [[11.94, 35.49, 6.55, 0, 47.96, -91.3], [9E9, 9E9, 9E9, 9E9, 9E9, 9E9]];
	VAR jointtarget CDP_2551 := [[12.01, 35.49, 6.56, 0, 47.96, -91.23], [9E9, 9E9, 9E9, 9E9, 9E9, 9E9]];
	VAR jointtarget CDP_2552 := [[12.08, 35.49, 6.56, 0, 47.95, -91.16], [9E9, 9E9, 9E9, 9E9, 9E9, 9E9]];
	VAR jointtarget CDP_2553 := [[12.15, 35.49, 6.56, 0, 47.95, -91.09], [9E9, 9E9, 9E9, 9E9, 9E9, 9E9]];
	VAR jointtarget CDP_2554 := [[12.21, 35.48, 6.56, 0, 47.95, -91.03], [9E9, 9E9, 9E9, 9E9, 9E9, 9E9]];
	VAR jointtarget CDP_2555 := [[12.28, 35.48, 6.57, 0, 47.95, -90.96], [9E9, 9E9, 9E9, 9E9, 9E9, 9E9]];
	VAR jointtarget CDP_2556 := [[12.35, 35.48, 6.57, 0, 47.95, -90.89], [9E9, 9E9, 9E9, 9E9, 9E9, 9E9]];
	VAR jointtarget CDP_2557 := [[12.42, 35.48, 6.57, 0, 47.95, -90.82], [9E9, 9E9, 9E9, 9E9, 9E9, 9E9]];
	VAR jointtarget CDP_2558 := [[12.49, 35.48, 6.57, 0, 47.95, -90.75], [9E9, 9E9, 9E9, 9E9, 9E9, 9E9]];
	VAR jointtarget CDP_2559 := [[12.55, 35.48, 6.57, 0, 47.95, -90.69], [9E9, 9E9, 9E9, 9E9, 9E9, 9E9]];
	VAR jointtarget CDP_2560 := [[12.69, 35.49, 6.55, 0, 47.96, -85.39], [9E9, 9E9, 9E9, 9E9, 9E9, 9E9]];
	VAR jointtarget CDP_2561 := [[12.81, 35.53, 6.49, 0, 47.98, -74.94], [9E9, 9E9, 9E9, 9E9, 9E9, 9E9]];
	VAR jointtarget CDP_2562 := [[12.93, 35.59, 6.39, 0, 48.03, -64.5], [9E9, 9E9, 9E9, 9E9, 9E9, 9E9]];
	VAR jointtarget CDP_2563 := [[13.04, 35.67, 6.24, 0, 48.09, -54.07], [9E9, 9E9, 9E9, 9E9, 9E9, 9E9]];
	VAR jointtarget CDP_2564 := [[13.13, 35.77, 6.07, 0, 48.16, -43.65], [9E9, 9E9, 9E9, 9E9, 9E9, 9E9]];
	VAR jointtarget CDP_2565 := [[13.2, 35.89, 5.86, 0, 48.24, -33.25], [9E9, 9E9, 9E9, 9E9, 9E9, 9E9]];
	VAR jointtarget CDP_2566 := [[13.25, 36.02, 5.64, 0, 48.34, -22.88], [9E9, 9E9, 9E9, 9E9, 9E9, 9E9]];
	VAR jointtarget CDP_2567 := [[13.28, 36.16, 5.4, 0, 48.44, -12.53], [9E9, 9E9, 9E9, 9E9, 9E9, 9E9]];
	VAR jointtarget CDP_2568 := [[13.29, 36.31, 5.15, 0, 48.54, -2.2], [9E9, 9E9, 9E9, 9E9, 9E9, 9E9]];
	VAR jointtarget CDP_2569 := [[13.27, 36.45, 4.91, 0, 48.64, 8.11], [9E9, 9E9, 9E9, 9E9, 9E9, 9E9]];
	VAR jointtarget CDP_2570 := [[13.23, 36.58, 4.68, 0, 48.74, 18.39], [9E9, 9E9, 9E9, 9E9, 9E9, 9E9]];
	VAR jointtarget CDP_2571 := [[13.17, 36.71, 4.46, 0, 48.83, 28.65], [9E9, 9E9, 9E9, 9E9, 9E9, 9E9]];
	VAR jointtarget CDP_2572 := [[13.08, 36.82, 4.27, 0, 48.91, 38.9], [9E9, 9E9, 9E9, 9E9, 9E9, 9E9]];
	VAR jointtarget CDP_2573 := [[12.99, 36.92, 4.11, 0, 48.98, 49.12], [9E9, 9E9, 9E9, 9E9, 9E9, 9E9]];
	VAR jointtarget CDP_2574 := [[12.88, 36.99, 3.98, 0, 49.03, 59.33], [9E9, 9E9, 9E9, 9E9, 9E9, 9E9]];
	VAR jointtarget CDP_2575 := [[12.75, 37.04, 3.89, 0, 49.07, 69.54], [9E9, 9E9, 9E9, 9E9, 9E9, 9E9]];
	VAR jointtarget CDP_2576 := [[12.63, 37.07, 3.85, 0, 49.09, 79.73], [9E9, 9E9, 9E9, 9E9, 9E9, 9E9]];
	VAR jointtarget CDP_2577 := [[12.5, 37.07, 3.85, 0, 49.09, 89.93], [9E9, 9E9, 9E9, 9E9, 9E9, 9E9]];
	VAR jointtarget CDP_2578 := [[12.37, 37.04, 3.89, 0, 49.07, 100.13], [9E9, 9E9, 9E9, 9E9, 9E9, 9E9]];
	VAR jointtarget CDP_2579 := [[12.25, 36.99, 3.98, 0, 49.03, 110.33], [9E9, 9E9, 9E9, 9E9, 9E9, 9E9]];
	VAR jointtarget CDP_2580 := [[12.19, 36.96, 4.03, 0, 49.01, 115.43], [9E9, 9E9, 9E9, 9E9, 9E9, 9E9]];
	VAR jointtarget CDP_2581 := [[12.13, 36.93, 4.09, 0, 48.98, 115.37], [9E9, 9E9, 9E9, 9E9, 9E9, 9E9]];
	VAR jointtarget CDP_2582 := [[12.07, 36.89, 4.14, 0, 48.96, 115.31], [9E9, 9E9, 9E9, 9E9, 9E9, 9E9]];
	VAR jointtarget CDP_2583 := [[12.01, 36.86, 4.2, 0, 48.94, 115.25], [9E9, 9E9, 9E9, 9E9, 9E9, 9E9]];
	VAR jointtarget CDP_2584 := [[11.95, 36.83, 4.25, 0, 48.92, 115.19], [9E9, 9E9, 9E9, 9E9, 9E9, 9E9]];
	VAR jointtarget CDP_2585 := [[11.89, 36.8, 4.31, 0, 48.89, 115.13], [9E9, 9E9, 9E9, 9E9, 9E9, 9E9]];
	VAR jointtarget CDP_2586 := [[11.83, 36.77, 4.36, 0, 48.87, 115.07], [9E9, 9E9, 9E9, 9E9, 9E9, 9E9]];
	VAR jointtarget CDP_2587 := [[11.77, 36.74, 4.41, 0, 48.85, 115.01], [9E9, 9E9, 9E9, 9E9, 9E9, 9E9]];
	VAR jointtarget CDP_2588 := [[11.71, 36.71, 4.47, 0, 48.83, 114.95], [9E9, 9E9, 9E9, 9E9, 9E9, 9E9]];
	VAR jointtarget CDP_2589 := [[11.65, 36.68, 4.52, 0, 48.8, 114.89], [9E9, 9E9, 9E9, 9E9, 9E9, 9E9]];
	VAR jointtarget CDP_2590 := [[11.59, 36.64, 4.57, 0, 48.78, 114.83], [9E9, 9E9, 9E9, 9E9, 9E9, 9E9]];
	VAR jointtarget CDP_2591 := [[11.53, 36.61, 4.63, 0, 48.76, 114.77], [9E9, 9E9, 9E9, 9E9, 9E9, 9E9]];
	VAR jointtarget CDP_2592 := [[11.47, 36.58, 4.68, 0, 48.74, 114.71], [9E9, 9E9, 9E9, 9E9, 9E9, 9E9]];
	VAR jointtarget CDP_2593 := [[11.4, 36.55, 4.73, 0, 48.71, 114.64], [9E9, 9E9, 9E9, 9E9, 9E9, 9E9]];
	VAR jointtarget CDP_2594 := [[11.34, 36.52, 4.79, 0, 48.69, 114.58], [9E9, 9E9, 9E9, 9E9, 9E9, 9E9]];
	VAR jointtarget CDP_2595 := [[11.28, 36.49, 4.84, 0, 48.67, 114.52], [9E9, 9E9, 9E9, 9E9, 9E9, 9E9]];
	VAR jointtarget CDP_2596 := [[11.22, 36.46, 4.89, 0, 48.65, 114.46], [9E9, 9E9, 9E9, 9E9, 9E9, 9E9]];
	VAR jointtarget CDP_2597 := [[11.16, 36.43, 4.94, 0, 48.63, 114.4], [9E9, 9E9, 9E9, 9E9, 9E9, 9E9]];
	VAR jointtarget CDP_2598 := [[11.1, 36.4, 5, 0, 48.6, 114.34], [9E9, 9E9, 9E9, 9E9, 9E9, 9E9]];
	VAR jointtarget CDP_2599 := [[11.04, 36.37, 5.05, 0, 48.58, 114.28], [9E9, 9E9, 9E9, 9E9, 9E9, 9E9]];
	VAR jointtarget CDP_2600 := [[11.02, 36.36, 5.06, 0, 48.58, 113.93], [9E9, 9E9, 9E9, 9E9, 9E9, 9E9]];
	VAR jointtarget CDP_2601 := [[11.01, 36.35, 5.07, 0, 48.57, 113.26], [9E9, 9E9, 9E9, 9E9, 9E9, 9E9]];
	VAR jointtarget CDP_2602 := [[10.99, 36.35, 5.09, 0, 48.57, 112.58], [9E9, 9E9, 9E9, 9E9, 9E9, 9E9]];
	VAR jointtarget CDP_2603 := [[10.98, 36.34, 5.1, 0, 48.56, 111.9], [9E9, 9E9, 9E9, 9E9, 9E9, 9E9]];
	VAR jointtarget CDP_2604 := [[10.96, 36.33, 5.11, 0, 48.56, 111.22], [9E9, 9E9, 9E9, 9E9, 9E9, 9E9]];
	VAR jointtarget CDP_2605 := [[10.95, 36.33, 5.12, 0, 48.55, 110.55], [9E9, 9E9, 9E9, 9E9, 9E9, 9E9]];
	VAR jointtarget CDP_2606 := [[10.93, 36.32, 5.13, 0, 48.55, 109.87], [9E9, 9E9, 9E9, 9E9, 9E9, 9E9]];
	VAR jointtarget CDP_2607 := [[10.91, 36.31, 5.14, 0, 48.54, 109.19], [9E9, 9E9, 9E9, 9E9, 9E9, 9E9]];
	VAR jointtarget CDP_2608 := [[10.9, 36.31, 5.15, 0, 48.54, 108.51], [9E9, 9E9, 9E9, 9E9, 9E9, 9E9]];
	VAR jointtarget CDP_2609 := [[10.88, 36.3, 5.16, 0, 48.54, 107.83], [9E9, 9E9, 9E9, 9E9, 9E9, 9E9]];
	VAR jointtarget CDP_2610 := [[10.87, 36.3, 5.17, 0, 48.53, 107.16], [9E9, 9E9, 9E9, 9E9, 9E9, 9E9]];
	VAR jointtarget CDP_2611 := [[10.85, 36.29, 5.18, 0, 48.53, 106.48], [9E9, 9E9, 9E9, 9E9, 9E9, 9E9]];
	VAR jointtarget CDP_2612 := [[10.83, 36.29, 5.19, 0, 48.53, 105.8], [9E9, 9E9, 9E9, 9E9, 9E9, 9E9]];
	VAR jointtarget CDP_2613 := [[10.82, 36.28, 5.2, 0, 48.52, 105.12], [9E9, 9E9, 9E9, 9E9, 9E9, 9E9]];
	VAR jointtarget CDP_2614 := [[10.8, 36.28, 5.2, 0, 48.52, 104.44], [9E9, 9E9, 9E9, 9E9, 9E9, 9E9]];
	VAR jointtarget CDP_2615 := [[10.79, 36.27, 5.21, 0, 48.52, 103.77], [9E9, 9E9, 9E9, 9E9, 9E9, 9E9]];
	VAR jointtarget CDP_2616 := [[10.77, 36.27, 5.22, 0, 48.51, 103.09], [9E9, 9E9, 9E9, 9E9, 9E9, 9E9]];
	VAR jointtarget CDP_2617 := [[10.75, 36.27, 5.22, 0, 48.51, 102.41], [9E9, 9E9, 9E9, 9E9, 9E9, 9E9]];
	VAR jointtarget CDP_2618 := [[10.74, 36.26, 5.23, 0, 48.51, 101.73], [9E9, 9E9, 9E9, 9E9, 9E9, 9E9]];
	VAR jointtarget CDP_2619 := [[10.72, 36.26, 5.24, 0, 48.5, 101.05], [9E9, 9E9, 9E9, 9E9, 9E9, 9E9]];
	VAR jointtarget CDP_2620 := [[9.64, 36.05, 5.6, 0, 48.35, 99.64], [9E9, 9E9, 9E9, 9E9, 9E9, 9E9]];
	VAR jointtarget CDP_2621 := [[8.56, 35.86, 5.92, 0, 48.22, 98.56], [9E9, 9E9, 9E9, 9E9, 9E9, 9E9]];
	VAR jointtarget CDP_2622 := [[7.47, 35.69, 6.21, 0, 48.1, 97.47], [9E9, 9E9, 9E9, 9E9, 9E9, 9E9]];
	VAR jointtarget CDP_2623 := [[6.38, 35.55, 6.45, 0, 48, 96.38], [9E9, 9E9, 9E9, 9E9, 9E9, 9E9]];
	VAR jointtarget CDP_2624 := [[5.28, 35.43, 6.66, 0, 47.91, 95.28], [9E9, 9E9, 9E9, 9E9, 9E9, 9E9]];
	VAR jointtarget CDP_2625 := [[4.17, 35.33, 6.82, 0, 47.84, 94.17], [9E9, 9E9, 9E9, 9E9, 9E9, 9E9]];
	VAR jointtarget CDP_2626 := [[3.07, 35.26, 6.95, 0, 47.79, 93.07], [9E9, 9E9, 9E9, 9E9, 9E9, 9E9]];
	VAR jointtarget CDP_2627 := [[1.96, 35.2, 7.04, 0, 47.76, 91.96], [9E9, 9E9, 9E9, 9E9, 9E9, 9E9]];
	VAR jointtarget CDP_2628 := [[0.85, 35.18, 7.09, 0, 47.73, 90.85], [9E9, 9E9, 9E9, 9E9, 9E9, 9E9]];
	VAR jointtarget CDP_2629 := [[-0.26, 35.17, 7.1, 0, 47.73, 89.74], [9E9, 9E9, 9E9, 9E9, 9E9, 9E9]];
	VAR jointtarget CDP_2630 := [[-1.37, 35.19, 7.07, 0, 47.74, 88.63], [9E9, 9E9, 9E9, 9E9, 9E9, 9E9]];
	VAR jointtarget CDP_2631 := [[-2.48, 35.23, 7, 0, 47.77, 87.52], [9E9, 9E9, 9E9, 9E9, 9E9, 9E9]];
	VAR jointtarget CDP_2632 := [[-3.59, 35.29, 6.9, 0, 47.82, 86.41], [9E9, 9E9, 9E9, 9E9, 9E9, 9E9]];
	VAR jointtarget CDP_2633 := [[-4.7, 35.38, 6.75, 0, 47.88, 85.3], [9E9, 9E9, 9E9, 9E9, 9E9, 9E9]];
	VAR jointtarget CDP_2634 := [[-5.8, 35.48, 6.56, 0, 47.95, 84.2], [9E9, 9E9, 9E9, 9E9, 9E9, 9E9]];
	VAR jointtarget CDP_2635 := [[-6.9, 35.62, 6.34, 0, 48.05, 83.1], [9E9, 9E9, 9E9, 9E9, 9E9, 9E9]];
	VAR jointtarget CDP_2636 := [[-7.99, 35.77, 6.08, 0, 48.16, 82.01], [9E9, 9E9, 9E9, 9E9, 9E9, 9E9]];
	VAR jointtarget CDP_2637 := [[-9.08, 35.95, 5.77, 0, 48.28, 80.92], [9E9, 9E9, 9E9, 9E9, 9E9, 9E9]];
	VAR jointtarget CDP_2638 := [[-10.16, 36.15, 5.43, 0, 48.42, 79.84], [9E9, 9E9, 9E9, 9E9, 9E9, 9E9]];
	VAR jointtarget CDP_2639 := [[-11.23, 36.37, 5.05, 0, 48.58, 78.77], [9E9, 9E9, 9E9, 9E9, 9E9, 9E9]];
	VAR jointtarget CDP_2640 := [[-11.28, 36.38, 5.03, 0, 48.59, 79.81], [9E9, 9E9, 9E9, 9E9, 9E9, 9E9]];
	VAR jointtarget CDP_2641 := [[-11.34, 36.39, 5.02, 0, 48.6, 81.95], [9E9, 9E9, 9E9, 9E9, 9E9, 9E9]];
	VAR jointtarget CDP_2642 := [[-11.39, 36.39, 5.01, 0, 48.6, 84.09], [9E9, 9E9, 9E9, 9E9, 9E9, 9E9]];
	VAR jointtarget CDP_2643 := [[-11.45, 36.4, 5, 0, 48.6, 86.23], [9E9, 9E9, 9E9, 9E9, 9E9, 9E9]];
	VAR jointtarget CDP_2644 := [[-11.5, 36.4, 5, 0, 48.6, 88.37], [9E9, 9E9, 9E9, 9E9, 9E9, 9E9]];
	VAR jointtarget CDP_2645 := [[-11.56, 36.4, 5, 0, 48.6, 90.51], [9E9, 9E9, 9E9, 9E9, 9E9, 9E9]];
	VAR jointtarget CDP_2646 := [[-11.61, 36.39, 5, 0, 48.6, 92.65], [9E9, 9E9, 9E9, 9E9, 9E9, 9E9]];
	VAR jointtarget CDP_2647 := [[-11.67, 36.39, 5.01, 0, 48.6, 94.78], [9E9, 9E9, 9E9, 9E9, 9E9, 9E9]];
	VAR jointtarget CDP_2648 := [[-11.72, 36.38, 5.03, 0, 48.59, 96.92], [9E9, 9E9, 9E9, 9E9, 9E9, 9E9]];
	VAR jointtarget CDP_2649 := [[-11.78, 36.37, 5.04, 0, 48.59, 99.06], [9E9, 9E9, 9E9, 9E9, 9E9, 9E9]];
	VAR jointtarget CDP_2650 := [[-11.83, 36.36, 5.06, 0, 48.58, 101.2], [9E9, 9E9, 9E9, 9E9, 9E9, 9E9]];
	VAR jointtarget CDP_2651 := [[-11.89, 36.35, 5.09, 0, 48.57, 103.34], [9E9, 9E9, 9E9, 9E9, 9E9, 9E9]];
	VAR jointtarget CDP_2652 := [[-11.94, 36.33, 5.11, 0, 48.56, 105.48], [9E9, 9E9, 9E9, 9E9, 9E9, 9E9]];
	VAR jointtarget CDP_2653 := [[-11.99, 36.31, 5.15, 0, 48.54, 107.63], [9E9, 9E9, 9E9, 9E9, 9E9, 9E9]];
	VAR jointtarget CDP_2654 := [[-12.04, 36.29, 5.18, 0, 48.53, 109.77], [9E9, 9E9, 9E9, 9E9, 9E9, 9E9]];
	VAR jointtarget CDP_2655 := [[-12.09, 36.27, 5.22, 0, 48.51, 111.91], [9E9, 9E9, 9E9, 9E9, 9E9, 9E9]];
	VAR jointtarget CDP_2656 := [[-12.15, 36.24, 5.26, 0, 48.49, 114.05], [9E9, 9E9, 9E9, 9E9, 9E9, 9E9]];
	VAR jointtarget CDP_2657 := [[-12.19, 36.22, 5.31, 0, 48.47, 116.2], [9E9, 9E9, 9E9, 9E9, 9E9, 9E9]];
	VAR jointtarget CDP_2658 := [[-12.24, 36.19, 5.36, 0, 48.45, 118.34], [9E9, 9E9, 9E9, 9E9, 9E9, 9E9]];
	VAR jointtarget CDP_2659 := [[-12.29, 36.16, 5.41, 0, 48.43, 120.49], [9E9, 9E9, 9E9, 9E9, 9E9, 9E9]];
	VAR jointtarget CDP_2660 := [[-12.32, 36.14, 5.44, 0, 48.42, 121.56], [9E9, 9E9, 9E9, 9E9, 9E9, 9E9]];
	VAR jointtarget CDP_2661 := [[-12.35, 36.12, 5.47, 0, 48.41, 121.53], [9E9, 9E9, 9E9, 9E9, 9E9, 9E9]];
	VAR jointtarget CDP_2662 := [[-12.38, 36.1, 5.51, 0, 48.39, 121.5], [9E9, 9E9, 9E9, 9E9, 9E9, 9E9]];
	VAR jointtarget CDP_2663 := [[-12.41, 36.08, 5.54, 0, 48.38, 121.47], [9E9, 9E9, 9E9, 9E9, 9E9, 9E9]];
	VAR jointtarget CDP_2664 := [[-12.43, 36.06, 5.57, 0, 48.36, 121.44], [9E9, 9E9, 9E9, 9E9, 9E9, 9E9]];
	VAR jointtarget CDP_2665 := [[-12.46, 36.04, 5.61, 0, 48.35, 121.41], [9E9, 9E9, 9E9, 9E9, 9E9, 9E9]];
	VAR jointtarget CDP_2666 := [[-12.49, 36.02, 5.64, 0, 48.34, 121.39], [9E9, 9E9, 9E9, 9E9, 9E9, 9E9]];
	VAR jointtarget CDP_2667 := [[-12.52, 36.01, 5.67, 0, 48.32, 121.36], [9E9, 9E9, 9E9, 9E9, 9E9, 9E9]];
	VAR jointtarget CDP_2668 := [[-12.55, 35.99, 5.7, 0, 48.31, 121.33], [9E9, 9E9, 9E9, 9E9, 9E9, 9E9]];
	VAR jointtarget CDP_2669 := [[-12.58, 35.97, 5.74, 0, 48.3, 121.3], [9E9, 9E9, 9E9, 9E9, 9E9, 9E9]];
	VAR jointtarget CDP_2670 := [[-12.61, 35.95, 5.77, 0, 48.28, 121.27], [9E9, 9E9, 9E9, 9E9, 9E9, 9E9]];
	VAR jointtarget CDP_2671 := [[-12.63, 35.93, 5.8, 0, 48.27, 121.24], [9E9, 9E9, 9E9, 9E9, 9E9, 9E9]];
	VAR jointtarget CDP_2672 := [[-12.66, 35.91, 5.83, 0, 48.26, 121.21], [9E9, 9E9, 9E9, 9E9, 9E9, 9E9]];
	VAR jointtarget CDP_2673 := [[-12.69, 35.89, 5.87, 0, 48.24, 121.18], [9E9, 9E9, 9E9, 9E9, 9E9, 9E9]];
	VAR jointtarget CDP_2674 := [[-12.72, 35.87, 5.9, 0, 48.23, 121.16], [9E9, 9E9, 9E9, 9E9, 9E9, 9E9]];
	VAR jointtarget CDP_2675 := [[-12.75, 35.85, 5.93, 0, 48.22, 121.13], [9E9, 9E9, 9E9, 9E9, 9E9, 9E9]];
	VAR jointtarget CDP_2676 := [[-12.78, 35.84, 5.96, 0, 48.2, 121.1], [9E9, 9E9, 9E9, 9E9, 9E9, 9E9]];
	VAR jointtarget CDP_2677 := [[-12.81, 35.82, 5.99, 0, 48.19, 121.07], [9E9, 9E9, 9E9, 9E9, 9E9, 9E9]];
	VAR jointtarget CDP_2678 := [[-12.84, 35.8, 6.03, 0, 48.18, 121.04], [9E9, 9E9, 9E9, 9E9, 9E9, 9E9]];
	VAR jointtarget CDP_2679 := [[-12.86, 35.78, 6.06, 0, 48.16, 121.01], [9E9, 9E9, 9E9, 9E9, 9E9, 9E9]];
	VAR jointtarget CDP_2680 := [[-13.02, 35.71, 6.18, 0, 48.11, 114.17], [9E9, 9E9, 9E9, 9E9, 9E9, 9E9]];
	VAR jointtarget CDP_2681 := [[-13.18, 35.67, 6.24, 0, 48.09, 100.62], [9E9, 9E9, 9E9, 9E9, 9E9, 9E9]];
	VAR jointtarget CDP_2682 := [[-13.34, 35.68, 6.22, 0, 48.09, 87.07], [9E9, 9E9, 9E9, 9E9, 9E9, 9E9]];
	VAR jointtarget CDP_2683 := [[-13.5, 35.73, 6.14, 0, 48.13, 73.52], [9E9, 9E9, 9E9, 9E9, 9E9, 9E9]];
	VAR jointtarget CDP_2684 := [[-13.64, 35.82, 5.99, 0, 48.19, 59.99], [9E9, 9E9, 9E9, 9E9, 9E9, 9E9]];
	VAR jointtarget CDP_2685 := [[-13.76, 35.94, 5.78, 0, 48.28, 46.48], [9E9, 9E9, 9E9, 9E9, 9E9, 9E9]];
	VAR jointtarget CDP_2686 := [[-13.85, 36.09, 5.52, 0, 48.39, 33.01], [9E9, 9E9, 9E9, 9E9, 9E9, 9E9]];
	VAR jointtarget CDP_2687 := [[-13.91, 36.26, 5.23, 0, 48.51, 19.56], [9E9, 9E9, 9E9, 9E9, 9E9, 9E9]];
	VAR jointtarget CDP_2688 := [[-13.92, 36.44, 4.93, 0, 48.63, 6.16], [9E9, 9E9, 9E9, 9E9, 9E9, 9E9]];
	VAR jointtarget CDP_2689 := [[-13.9, 36.62, 4.62, 0, 48.76, -7.21], [9E9, 9E9, 9E9, 9E9, 9E9, 9E9]];
	VAR jointtarget CDP_2690 := [[-13.85, 36.79, 4.33, 0, 48.88, -20.54], [9E9, 9E9, 9E9, 9E9, 9E9, 9E9]];
	VAR jointtarget CDP_2691 := [[-13.76, 36.93, 4.07, 0, 48.99, -33.84], [9E9, 9E9, 9E9, 9E9, 9E9, 9E9]];
	VAR jointtarget CDP_2692 := [[-13.64, 37.06, 3.86, 0, 49.08, -47.11], [9E9, 9E9, 9E9, 9E9, 9E9, 9E9]];
	VAR jointtarget CDP_2693 := [[-13.5, 37.15, 3.71, 0, 49.14, -60.35], [9E9, 9E9, 9E9, 9E9, 9E9, 9E9]];
	VAR jointtarget CDP_2694 := [[-13.34, 37.2, 3.62, 0, 49.18, -73.59], [9E9, 9E9, 9E9, 9E9, 9E9, 9E9]];
	VAR jointtarget CDP_2695 := [[-13.18, 37.21, 3.61, 0, 49.19, -86.81], [9E9, 9E9, 9E9, 9E9, 9E9, 9E9]];
	VAR jointtarget CDP_2696 := [[-13.02, 37.17, 3.66, 0, 49.16, -100.04], [9E9, 9E9, 9E9, 9E9, 9E9, 9E9]];
	VAR jointtarget CDP_2697 := [[-12.88, 37.1, 3.78, 0, 49.11, -113.28], [9E9, 9E9, 9E9, 9E9, 9E9, 9E9]];
	VAR jointtarget CDP_2698 := [[-12.75, 37, 3.97, 0, 49.03, -126.54], [9E9, 9E9, 9E9, 9E9, 9E9, 9E9]];
	VAR jointtarget CDP_2699 := [[-12.64, 36.86, 4.21, 0, 48.94, -139.82], [9E9, 9E9, 9E9, 9E9, 9E9, 9E9]];
	VAR jointtarget CDP_2700 := [[-12.62, 36.82, 4.28, 0, 48.91, -146.49], [9E9, 9E9, 9E9, 9E9, 9E9, 9E9]];
	VAR jointtarget CDP_2701 := [[-12.59, 36.78, 4.35, 0, 48.88, -146.47], [9E9, 9E9, 9E9, 9E9, 9E9, 9E9]];
	VAR jointtarget CDP_2702 := [[-12.57, 36.73, 4.42, 0, 48.85, -146.44], [9E9, 9E9, 9E9, 9E9, 9E9, 9E9]];
	VAR jointtarget CDP_2703 := [[-12.54, 36.69, 4.49, 0, 48.82, -146.42], [9E9, 9E9, 9E9, 9E9, 9E9, 9E9]];
	VAR jointtarget CDP_2704 := [[-12.52, 36.65, 4.56, 0, 48.79, -146.4], [9E9, 9E9, 9E9, 9E9, 9E9, 9E9]];
	VAR jointtarget CDP_2705 := [[-12.49, 36.61, 4.63, 0, 48.76, -146.37], [9E9, 9E9, 9E9, 9E9, 9E9, 9E9]];
	VAR jointtarget CDP_2706 := [[-12.47, 36.57, 4.7, 0, 48.73, -146.35], [9E9, 9E9, 9E9, 9E9, 9E9, 9E9]];
	VAR jointtarget CDP_2707 := [[-12.44, 36.53, 4.77, 0, 48.7, -146.32], [9E9, 9E9, 9E9, 9E9, 9E9, 9E9]];
	VAR jointtarget CDP_2708 := [[-12.42, 36.49, 4.84, 0, 48.67, -146.3], [9E9, 9E9, 9E9, 9E9, 9E9, 9E9]];
	VAR jointtarget CDP_2709 := [[-12.39, 36.45, 4.91, 0, 48.64, -146.27], [9E9, 9E9, 9E9, 9E9, 9E9, 9E9]];
	VAR jointtarget CDP_2710 := [[-12.37, 36.41, 4.98, 0, 48.61, -146.25], [9E9, 9E9, 9E9, 9E9, 9E9, 9E9]];
	VAR jointtarget CDP_2711 := [[-12.34, 36.36, 5.05, 0, 48.58, -146.22], [9E9, 9E9, 9E9, 9E9, 9E9, 9E9]];
	VAR jointtarget CDP_2712 := [[-12.32, 36.32, 5.13, 0, 48.55, -146.2], [9E9, 9E9, 9E9, 9E9, 9E9, 9E9]];
	VAR jointtarget CDP_2713 := [[-12.29, 36.28, 5.2, 0, 48.52, -146.17], [9E9, 9E9, 9E9, 9E9, 9E9, 9E9]];
	VAR jointtarget CDP_2714 := [[-12.27, 36.24, 5.27, 0, 48.49, -146.15], [9E9, 9E9, 9E9, 9E9, 9E9, 9E9]];
	VAR jointtarget CDP_2715 := [[-12.24, 36.2, 5.34, 0, 48.46, -146.12], [9E9, 9E9, 9E9, 9E9, 9E9, 9E9]];
	VAR jointtarget CDP_2716 := [[-12.22, 36.16, 5.41, 0, 48.43, -146.1], [9E9, 9E9, 9E9, 9E9, 9E9, 9E9]];
	VAR jointtarget CDP_2717 := [[-12.19, 36.12, 5.48, 0, 48.4, -146.07], [9E9, 9E9, 9E9, 9E9, 9E9, 9E9]];
	VAR jointtarget CDP_2718 := [[-12.17, 36.08, 5.55, 0, 48.38, -146.05], [9E9, 9E9, 9E9, 9E9, 9E9, 9E9]];
	VAR jointtarget CDP_2719 := [[-12.14, 36.04, 5.62, 0, 48.35, -146.02], [9E9, 9E9, 9E9, 9E9, 9E9, 9E9]];
	VAR jointtarget CDP_2720 := [[-12.14, 36.03, 5.64, 0, 48.34, -145.46], [9E9, 9E9, 9E9, 9E9, 9E9, 9E9]];
	VAR jointtarget CDP_2721 := [[-12.13, 36.01, 5.66, 0, 48.33, -144.35], [9E9, 9E9, 9E9, 9E9, 9E9, 9E9]];
	VAR jointtarget CDP_2722 := [[-12.12, 36, 5.68, 0, 48.32, -143.24], [9E9, 9E9, 9E9, 9E9, 9E9, 9E9]];
	VAR jointtarget CDP_2723 := [[-12.11, 35.99, 5.7, 0, 48.31, -142.13], [9E9, 9E9, 9E9, 9E9, 9E9, 9E9]];
	VAR jointtarget CDP_2724 := [[-12.1, 35.98, 5.72, 0, 48.3, -141.01], [9E9, 9E9, 9E9, 9E9, 9E9, 9E9]];
	VAR jointtarget CDP_2725 := [[-12.09, 35.96, 5.74, 0, 48.3, -139.9], [9E9, 9E9, 9E9, 9E9, 9E9, 9E9]];
	VAR jointtarget CDP_2726 := [[-12.08, 35.95, 5.76, 0, 48.29, -138.79], [9E9, 9E9, 9E9, 9E9, 9E9, 9E9]];
	VAR jointtarget CDP_2727 := [[-12.07, 35.94, 5.78, 0, 48.28, -137.68], [9E9, 9E9, 9E9, 9E9, 9E9, 9E9]];
	VAR jointtarget CDP_2728 := [[-12.06, 35.93, 5.8, 0, 48.27, -136.56], [9E9, 9E9, 9E9, 9E9, 9E9, 9E9]];
	VAR jointtarget CDP_2729 := [[-12.05, 35.92, 5.82, 0, 48.26, -135.45], [9E9, 9E9, 9E9, 9E9, 9E9, 9E9]];
	VAR jointtarget CDP_2730 := [[-12.04, 35.91, 5.83, 0, 48.26, -134.34], [9E9, 9E9, 9E9, 9E9, 9E9, 9E9]];
	VAR jointtarget CDP_2731 := [[-12.03, 35.9, 5.85, 0, 48.25, -133.22], [9E9, 9E9, 9E9, 9E9, 9E9, 9E9]];
	VAR jointtarget CDP_2732 := [[-12.02, 35.89, 5.87, 0, 48.24, -132.11], [9E9, 9E9, 9E9, 9E9, 9E9, 9E9]];
	VAR jointtarget CDP_2733 := [[-12.01, 35.88, 5.89, 0, 48.24, -130.99], [9E9, 9E9, 9E9, 9E9, 9E9, 9E9]];
	VAR jointtarget CDP_2734 := [[-12, 35.87, 5.9, 0, 48.23, -129.88], [9E9, 9E9, 9E9, 9E9, 9E9, 9E9]];
	VAR jointtarget CDP_2735 := [[-11.99, 35.86, 5.92, 0, 48.22, -128.76], [9E9, 9E9, 9E9, 9E9, 9E9, 9E9]];
	VAR jointtarget CDP_2736 := [[-11.98, 35.85, 5.94, 0, 48.22, -127.65], [9E9, 9E9, 9E9, 9E9, 9E9, 9E9]];
	VAR jointtarget CDP_2737 := [[-11.97, 35.84, 5.95, 0, 48.21, -126.53], [9E9, 9E9, 9E9, 9E9, 9E9, 9E9]];
	VAR jointtarget CDP_2738 := [[-11.96, 35.83, 5.97, 0, 48.21, -125.42], [9E9, 9E9, 9E9, 9E9, 9E9, 9E9]];
	VAR jointtarget CDP_2739 := [[-11.95, 35.82, 5.98, 0, 48.2, -124.3], [9E9, 9E9, 9E9, 9E9, 9E9, 9E9]];
	VAR jointtarget CDP_2740 := [[-11.94, 35.81, 5.99, 0, 48.2, -123.74], [9E9, 9E9, 9E9, 9E9, 9E9, 9E9]];
	VAR jointtarget CDP_2741 := [[-11.93, 35.8, 6.01, 0, 48.19, -123.73], [9E9, 9E9, 9E9, 9E9, 9E9, 9E9]];
	VAR jointtarget CDP_2742 := [[-11.92, 35.8, 6.02, 0, 48.19, -123.72], [9E9, 9E9, 9E9, 9E9, 9E9, 9E9]];
	VAR jointtarget CDP_2743 := [[-11.9, 35.79, 6.03, 0, 48.18, -123.71], [9E9, 9E9, 9E9, 9E9, 9E9, 9E9]];
	VAR jointtarget CDP_2744 := [[-11.89, 35.78, 6.04, 0, 48.18, -123.7], [9E9, 9E9, 9E9, 9E9, 9E9, 9E9]];
	VAR jointtarget CDP_2745 := [[-11.88, 35.77, 6.06, 0, 48.17, -123.69], [9E9, 9E9, 9E9, 9E9, 9E9, 9E9]];
	VAR jointtarget CDP_2746 := [[-11.87, 35.76, 6.07, 0, 48.17, -123.68], [9E9, 9E9, 9E9, 9E9, 9E9, 9E9]];
	VAR jointtarget CDP_2747 := [[-11.86, 35.76, 6.08, 0, 48.16, -123.66], [9E9, 9E9, 9E9, 9E9, 9E9, 9E9]];
	VAR jointtarget CDP_2748 := [[-11.85, 35.75, 6.1, 0, 48.16, -123.65], [9E9, 9E9, 9E9, 9E9, 9E9, 9E9]];
	VAR jointtarget CDP_2749 := [[-11.84, 35.74, 6.11, 0, 48.15, -123.64], [9E9, 9E9, 9E9, 9E9, 9E9, 9E9]];
	VAR jointtarget CDP_2750 := [[-11.83, 35.73, 6.12, 0, 48.15, -123.63], [9E9, 9E9, 9E9, 9E9, 9E9, 9E9]];
	VAR jointtarget CDP_2751 := [[-11.82, 35.72, 6.13, 0, 48.14, -123.62], [9E9, 9E9, 9E9, 9E9, 9E9, 9E9]];
	VAR jointtarget CDP_2752 := [[-11.81, 35.72, 6.15, 0, 48.14, -123.61], [9E9, 9E9, 9E9, 9E9, 9E9, 9E9]];
	VAR jointtarget CDP_2753 := [[-11.8, 35.71, 6.16, 0, 48.13, -123.6], [9E9, 9E9, 9E9, 9E9, 9E9, 9E9]];
	VAR jointtarget CDP_2754 := [[-11.79, 35.7, 6.17, 0, 48.13, -123.59], [9E9, 9E9, 9E9, 9E9, 9E9, 9E9]];
	VAR jointtarget CDP_2755 := [[-11.78, 35.69, 6.18, 0, 48.12, -123.58], [9E9, 9E9, 9E9, 9E9, 9E9, 9E9]];
	VAR jointtarget CDP_2756 := [[-11.77, 35.69, 6.2, 0, 48.12, -123.57], [9E9, 9E9, 9E9, 9E9, 9E9, 9E9]];
	VAR jointtarget CDP_2757 := [[-11.76, 35.68, 6.21, 0, 48.11, -123.56], [9E9, 9E9, 9E9, 9E9, 9E9, 9E9]];
	VAR jointtarget CDP_2758 := [[-11.75, 35.67, 6.22, 0, 48.11, -123.55], [9E9, 9E9, 9E9, 9E9, 9E9, 9E9]];
	VAR jointtarget CDP_2759 := [[-11.74, 35.66, 6.23, 0, 48.1, -123.54], [9E9, 9E9, 9E9, 9E9, 9E9, 9E9]];
	VAR jointtarget CDP_2760 := [[-10.65, 35.43, 6.63, 0, 47.94, -100.65], [9E9, 9E9, 9E9, 9E9, 9E9, 9E9]];
	VAR jointtarget CDP_2761 := [[-9.55, 35.22, 6.99, 0, 47.79, -99.55], [9E9, 9E9, 9E9, 9E9, 9E9, 9E9]];
	VAR jointtarget CDP_2762 := [[-8.44, 35.03, 7.31, 0, 47.66, -98.44], [9E9, 9E9, 9E9, 9E9, 9E9, 9E9]];
	VAR jointtarget CDP_2763 := [[-7.33, 34.87, 7.59, 0, 47.54, -97.33], [9E9, 9E9, 9E9, 9E9, 9E9, 9E9]];
	VAR jointtarget CDP_2764 := [[-6.21, 34.73, 7.82, 0, 47.45, -96.21], [9E9, 9E9, 9E9, 9E9, 9E9, 9E9]];
	VAR jointtarget CDP_2765 := [[-5.09, 34.61, 8.02, 0, 47.36, -95.09], [9E9, 9E9, 9E9, 9E9, 9E9, 9E9]];
	VAR jointtarget CDP_2766 := [[-3.96, 34.52, 8.18, 0, 47.3, -93.96], [9E9, 9E9, 9E9, 9E9, 9E9, 9E9]];
	VAR jointtarget CDP_2767 := [[-2.83, 34.45, 8.3, 0, 47.25, -92.83], [9E9, 9E9, 9E9, 9E9, 9E9, 9E9]];
	VAR jointtarget CDP_2768 := [[-1.7, 34.4, 8.38, 0, 47.22, -91.7], [9E9, 9E9, 9E9, 9E9, 9E9, 9E9]];
	VAR jointtarget CDP_2769 := [[-0.56, 34.38, 8.42, 0, 47.2, -90.56], [9E9, 9E9, 9E9, 9E9, 9E9, 9E9]];
	VAR jointtarget CDP_2770 := [[0.57, 34.38, 8.42, 0, 47.2, -89.43], [9E9, 9E9, 9E9, 9E9, 9E9, 9E9]];
	VAR jointtarget CDP_2771 := [[1.7, 34.4, 8.38, 0, 47.22, -88.3], [9E9, 9E9, 9E9, 9E9, 9E9, 9E9]];
	VAR jointtarget CDP_2772 := [[2.84, 34.45, 8.3, 0, 47.25, -87.16], [9E9, 9E9, 9E9, 9E9, 9E9, 9E9]];
	VAR jointtarget CDP_2773 := [[3.97, 34.52, 8.18, 0, 47.3, -86.03], [9E9, 9E9, 9E9, 9E9, 9E9, 9E9]];
	VAR jointtarget CDP_2774 := [[5.09, 34.61, 8.02, 0, 47.36, -84.91], [9E9, 9E9, 9E9, 9E9, 9E9, 9E9]];
	VAR jointtarget CDP_2775 := [[6.22, 34.73, 7.82, 0, 47.45, -83.78], [9E9, 9E9, 9E9, 9E9, 9E9, 9E9]];
	VAR jointtarget CDP_2776 := [[7.34, 34.87, 7.58, 0, 47.55, -82.66], [9E9, 9E9, 9E9, 9E9, 9E9, 9E9]];
	VAR jointtarget CDP_2777 := [[8.45, 35.03, 7.31, 0, 47.66, -81.55], [9E9, 9E9, 9E9, 9E9, 9E9, 9E9]];
	VAR jointtarget CDP_2778 := [[9.56, 35.22, 6.99, 0, 47.79, -80.44], [9E9, 9E9, 9E9, 9E9, 9E9, 9E9]];
	VAR jointtarget CDP_2779 := [[10.65, 35.43, 6.63, 0, 47.94, -79.35], [9E9, 9E9, 9E9, 9E9, 9E9, 9E9]];
	VAR jointtarget CDP_2780 := [[10.71, 35.44, 6.61, 0, 47.95, -78.19], [9E9, 9E9, 9E9, 9E9, 9E9, 9E9]];
	VAR jointtarget CDP_2781 := [[10.76, 35.46, 6.58, 0, 47.96, -75.95], [9E9, 9E9, 9E9, 9E9, 9E9, 9E9]];
	VAR jointtarget CDP_2782 := [[10.82, 35.47, 6.55, 0, 47.97, -73.7], [9E9, 9E9, 9E9, 9E9, 9E9, 9E9]];
	VAR jointtarget CDP_2783 := [[10.87, 35.49, 6.52, 0, 47.98, -71.45], [9E9, 9E9, 9E9, 9E9, 9E9, 9E9]];
	VAR jointtarget CDP_2784 := [[10.92, 35.52, 6.49, 0, 48, -69.2], [9E9, 9E9, 9E9, 9E9, 9E9, 9E9]];
	VAR jointtarget CDP_2785 := [[10.97, 35.54, 6.45, 0, 48.02, -66.96], [9E9, 9E9, 9E9, 9E9, 9E9, 9E9]];
	VAR jointtarget CDP_2786 := [[11.03, 35.56, 6.4, 0, 48.03, -64.72], [9E9, 9E9, 9E9, 9E9, 9E9, 9E9]];
	VAR jointtarget CDP_2787 := [[11.07, 35.59, 6.35, 0, 48.05, -62.47], [9E9, 9E9, 9E9, 9E9, 9E9, 9E9]];
	VAR jointtarget CDP_2788 := [[11.12, 35.62, 6.3, 0, 48.08, -60.23], [9E9, 9E9, 9E9, 9E9, 9E9, 9E9]];
	VAR jointtarget CDP_2789 := [[11.17, 35.65, 6.25, 0, 48.1, -57.99], [9E9, 9E9, 9E9, 9E9, 9E9, 9E9]];
	VAR jointtarget CDP_2790 := [[11.22, 35.69, 6.19, 0, 48.12, -55.75], [9E9, 9E9, 9E9, 9E9, 9E9, 9E9]];
	VAR jointtarget CDP_2791 := [[11.26, 35.72, 6.13, 0, 48.15, -53.51], [9E9, 9E9, 9E9, 9E9, 9E9, 9E9]];
	VAR jointtarget CDP_2792 := [[11.3, 35.76, 6.06, 0, 48.17, -51.27], [9E9, 9E9, 9E9, 9E9, 9E9, 9E9]];
	VAR jointtarget CDP_2793 := [[11.35, 35.8, 6, 0, 48.2, -49.04], [9E9, 9E9, 9E9, 9E9, 9E9, 9E9]];
	VAR jointtarget CDP_2794 := [[11.39, 35.84, 5.93, 0, 48.23, -46.8], [9E9, 9E9, 9E9, 9E9, 9E9, 9E9]];
	VAR jointtarget CDP_2795 := [[11.43, 35.88, 5.85, 0, 48.26, -44.57], [9E9, 9E9, 9E9, 9E9, 9E9, 9E9]];
	VAR jointtarget CDP_2796 := [[11.46, 35.93, 5.78, 0, 48.29, -42.34], [9E9, 9E9, 9E9, 9E9, 9E9, 9E9]];
	VAR jointtarget CDP_2797 := [[11.5, 35.98, 5.7, 0, 48.33, -40.11], [9E9, 9E9, 9E9, 9E9, 9E9, 9E9]];
	VAR jointtarget CDP_2798 := [[11.53, 36.02, 5.62, 0, 48.36, -37.88], [9E9, 9E9, 9E9, 9E9, 9E9, 9E9]];
	VAR jointtarget CDP_2799 := [[11.57, 36.07, 5.53, 0, 48.4, -35.65], [9E9, 9E9, 9E9, 9E9, 9E9, 9E9]];
	VAR jointtarget CDP_2800 := [[11.59, 36.1, 5.48, 0, 48.42, -34.54], [9E9, 9E9, 9E9, 9E9, 9E9, 9E9]];
	VAR jointtarget CDP_2801 := [[11.6, 36.13, 5.43, 0, 48.44, -34.52], [9E9, 9E9, 9E9, 9E9, 9E9, 9E9]];
	VAR jointtarget CDP_2802 := [[11.62, 36.16, 5.38, 0, 48.46, -34.5], [9E9, 9E9, 9E9, 9E9, 9E9, 9E9]];
	VAR jointtarget CDP_2803 := [[11.64, 36.19, 5.33, 0, 48.48, -34.48], [9E9, 9E9, 9E9, 9E9, 9E9, 9E9]];
	VAR jointtarget CDP_2804 := [[11.66, 36.22, 5.27, 0, 48.5, -34.46], [9E9, 9E9, 9E9, 9E9, 9E9, 9E9]];
	VAR jointtarget CDP_2805 := [[11.68, 36.25, 5.22, 0, 48.52, -34.44], [9E9, 9E9, 9E9, 9E9, 9E9, 9E9]];
	VAR jointtarget CDP_2806 := [[11.7, 36.28, 5.17, 0, 48.55, -34.42], [9E9, 9E9, 9E9, 9E9, 9E9, 9E9]];
	VAR jointtarget CDP_2807 := [[11.72, 36.31, 5.12, 0, 48.57, -34.41], [9E9, 9E9, 9E9, 9E9, 9E9, 9E9]];
	VAR jointtarget CDP_2808 := [[11.74, 36.34, 5.07, 0, 48.59, -34.39], [9E9, 9E9, 9E9, 9E9, 9E9, 9E9]];
	VAR jointtarget CDP_2809 := [[11.76, 36.37, 5.02, 0, 48.61, -34.37], [9E9, 9E9, 9E9, 9E9, 9E9, 9E9]];
	VAR jointtarget CDP_2810 := [[11.77, 36.4, 4.96, 0, 48.63, -34.35], [9E9, 9E9, 9E9, 9E9, 9E9, 9E9]];
	VAR jointtarget CDP_2811 := [[11.79, 36.43, 4.91, 0, 48.65, -34.33], [9E9, 9E9, 9E9, 9E9, 9E9, 9E9]];
	VAR jointtarget CDP_2812 := [[11.81, 36.46, 4.86, 0, 48.68, -34.31], [9E9, 9E9, 9E9, 9E9, 9E9, 9E9]];
	VAR jointtarget CDP_2813 := [[11.83, 36.49, 4.81, 0, 48.7, -34.29], [9E9, 9E9, 9E9, 9E9, 9E9, 9E9]];
	VAR jointtarget CDP_2814 := [[11.85, 36.52, 4.76, 0, 48.72, -34.27], [9E9, 9E9, 9E9, 9E9, 9E9, 9E9]];
	VAR jointtarget CDP_2815 := [[11.87, 36.56, 4.7, 0, 48.74, -34.26], [9E9, 9E9, 9E9, 9E9, 9E9, 9E9]];
	VAR jointtarget CDP_2816 := [[11.89, 36.59, 4.65, 0, 48.76, -34.24], [9E9, 9E9, 9E9, 9E9, 9E9, 9E9]];
	VAR jointtarget CDP_2817 := [[11.91, 36.62, 4.6, 0, 48.79, -34.22], [9E9, 9E9, 9E9, 9E9, 9E9, 9E9]];
	VAR jointtarget CDP_2818 := [[11.92, 36.65, 4.55, 0, 48.81, -34.2], [9E9, 9E9, 9E9, 9E9, 9E9, 9E9]];
	VAR jointtarget CDP_2819 := [[11.94, 36.68, 4.49, 0, 48.83, -34.18], [9E9, 9E9, 9E9, 9E9, 9E9, 9E9]];
	VAR jointtarget CDP_2820 := [[12.05, 36.81, 4.26, 0, 48.93, -40.77], [9E9, 9E9, 9E9, 9E9, 9E9, 9E9]];
	VAR jointtarget CDP_2821 := [[12.18, 36.92, 4.08, 0, 49, -54.03], [9E9, 9E9, 9E9, 9E9, 9E9, 9E9]];
	VAR jointtarget CDP_2822 := [[12.33, 36.99, 3.96, 0, 49.05, -67.26], [9E9, 9E9, 9E9, 9E9, 9E9, 9E9]];
	VAR jointtarget CDP_2823 := [[12.49, 37.02, 3.91, 0, 49.07, -80.49], [9E9, 9E9, 9E9, 9E9, 9E9, 9E9]];
	VAR jointtarget CDP_2824 := [[12.65, 37, 3.93, 0, 49.07, -93.72], [9E9, 9E9, 9E9, 9E9, 9E9, 9E9]];
	VAR jointtarget CDP_2825 := [[12.8, 36.95, 4.02, 0, 49.03, -106.95], [9E9, 9E9, 9E9, 9E9, 9E9, 9E9]];
	VAR jointtarget CDP_2826 := [[12.94, 36.86, 4.18, 0, 48.96, -120.2], [9E9, 9E9, 9E9, 9E9, 9E9, 9E9]];
	VAR jointtarget CDP_2827 := [[13.06, 36.74, 4.39, 0, 48.87, -133.47], [9E9, 9E9, 9E9, 9E9, 9E9, 9E9]];
	VAR jointtarget CDP_2828 := [[13.15, 36.59, 4.65, 0, 48.76, -146.77], [9E9, 9E9, 9E9, 9E9, 9E9, 9E9]];
	VAR jointtarget CDP_2829 := [[13.2, 36.42, 4.94, 0, 48.64, -160.1], [9E9, 9E9, 9E9, 9E9, 9E9, 9E9]];
	VAR jointtarget CDP_2830 := [[13.22, 36.24, 5.24, 0, 48.52, -173.47], [9E9, 9E9, 9E9, 9E9, 9E9, 9E9]];
	VAR jointtarget CDP_2831 := [[13.2, 36.06, 5.55, 0, 48.39, -186.88], [9E9, 9E9, 9E9, 9E9, 9E9, 9E9]];
	VAR jointtarget CDP_2832 := [[13.15, 35.9, 5.83, 0, 48.27, -200.32], [9E9, 9E9, 9E9, 9E9, 9E9, 9E9]];
	VAR jointtarget CDP_2833 := [[13.06, 35.75, 6.09, 0, 48.16, -213.8], [9E9, 9E9, 9E9, 9E9, 9E9, 9E9]];
	VAR jointtarget CDP_2834 := [[12.93, 35.63, 6.29, 0, 48.08, -227.31], [9E9, 9E9, 9E9, 9E9, 9E9, 9E9]];
	VAR jointtarget CDP_2835 := [[12.79, 35.54, 6.44, 0, 48.02, -240.84], [9E9, 9E9, 9E9, 9E9, 9E9, 9E9]];
	VAR jointtarget CDP_2836 := [[12.63, 35.49, 6.52, 0, 47.98, -254.39], [9E9, 9E9, 9E9, 9E9, 9E9, 9E9]];
	VAR jointtarget CDP_2837 := [[12.47, 35.49, 6.54, 0, 47.98, -267.94], [9E9, 9E9, 9E9, 9E9, 9E9, 9E9]];
	VAR jointtarget CDP_2838 := [[12.3, 35.52, 6.48, 0, 48, -281.49], [9E9, 9E9, 9E9, 9E9, 9E9, 9E9]];
	VAR jointtarget CDP_2839 := [[12.15, 35.6, 6.35, 0, 48.06, -295.03], [9E9, 9E9, 9E9, 9E9, 9E9, 9E9]];
	VAR jointtarget CDP_2840 := [[12.13, 35.62, 6.31, 0, 48.07, -301.75], [9E9, 9E9, 9E9, 9E9, 9E9, 9E9]];
	VAR jointtarget CDP_2841 := [[12.1, 35.63, 6.28, 0, 48.08, -301.78], [9E9, 9E9, 9E9, 9E9, 9E9, 9E9]];
	VAR jointtarget CDP_2842 := [[12.07, 35.65, 6.25, 0, 48.1, -301.81], [9E9, 9E9, 9E9, 9E9, 9E9, 9E9]];
	VAR jointtarget CDP_2843 := [[12.04, 35.67, 6.22, 0, 48.11, -301.84], [9E9, 9E9, 9E9, 9E9, 9E9, 9E9]];
	VAR jointtarget CDP_2844 := [[12.01, 35.69, 6.18, 0, 48.12, -301.87], [9E9, 9E9, 9E9, 9E9, 9E9, 9E9]];
	VAR jointtarget CDP_2845 := [[11.98, 35.71, 6.15, 0, 48.14, -301.89], [9E9, 9E9, 9E9, 9E9, 9E9, 9E9]];
	VAR jointtarget CDP_2846 := [[11.95, 35.73, 6.12, 0, 48.15, -301.92], [9E9, 9E9, 9E9, 9E9, 9E9, 9E9]];
	VAR jointtarget CDP_2847 := [[11.92, 35.75, 6.08, 0, 48.17, -301.95], [9E9, 9E9, 9E9, 9E9, 9E9, 9E9]];
	VAR jointtarget CDP_2848 := [[11.9, 35.77, 6.05, 0, 48.18, -301.98], [9E9, 9E9, 9E9, 9E9, 9E9, 9E9]];
	VAR jointtarget CDP_2849 := [[11.87, 35.79, 6.02, 0, 48.19, -302.01], [9E9, 9E9, 9E9, 9E9, 9E9, 9E9]];
	VAR jointtarget CDP_2850 := [[11.84, 35.81, 5.99, 0, 48.21, -302.04], [9E9, 9E9, 9E9, 9E9, 9E9, 9E9]];
	VAR jointtarget CDP_2851 := [[11.81, 35.83, 5.95, 0, 48.22, -302.07], [9E9, 9E9, 9E9, 9E9, 9E9, 9E9]];
	VAR jointtarget CDP_2852 := [[11.78, 35.85, 5.92, 0, 48.23, -302.09], [9E9, 9E9, 9E9, 9E9, 9E9, 9E9]];
	VAR jointtarget CDP_2853 := [[11.75, 35.87, 5.89, 0, 48.25, -302.12], [9E9, 9E9, 9E9, 9E9, 9E9, 9E9]];
	VAR jointtarget CDP_2854 := [[11.73, 35.88, 5.85, 0, 48.26, -302.15], [9E9, 9E9, 9E9, 9E9, 9E9, 9E9]];
	VAR jointtarget CDP_2855 := [[11.7, 35.9, 5.82, 0, 48.28, -302.18], [9E9, 9E9, 9E9, 9E9, 9E9, 9E9]];
	VAR jointtarget CDP_2856 := [[11.67, 35.92, 5.79, 0, 48.29, -302.21], [9E9, 9E9, 9E9, 9E9, 9E9, 9E9]];
	VAR jointtarget CDP_2857 := [[11.64, 35.94, 5.75, 0, 48.3, -302.24], [9E9, 9E9, 9E9, 9E9, 9E9, 9E9]];
	VAR jointtarget CDP_2858 := [[11.61, 35.96, 5.72, 0, 48.32, -302.27], [9E9, 9E9, 9E9, 9E9, 9E9, 9E9]];
	VAR jointtarget CDP_2859 := [[11.58, 35.98, 5.69, 0, 48.33, -302.29], [9E9, 9E9, 9E9, 9E9, 9E9, 9E9]];
	VAR jointtarget CDP_2860 := [[11.54, 36.01, 5.63, 0, 48.35, -301.24], [9E9, 9E9, 9E9, 9E9, 9E9, 9E9]];
	VAR jointtarget CDP_2861 := [[11.49, 36.04, 5.58, 0, 48.37, -299.1], [9E9, 9E9, 9E9, 9E9, 9E9, 9E9]];
	VAR jointtarget CDP_2862 := [[11.44, 36.07, 5.54, 0, 48.39, -296.95], [9E9, 9E9, 9E9, 9E9, 9E9, 9E9]];
	VAR jointtarget CDP_2863 := [[11.39, 36.1, 5.49, 0, 48.41, -294.81], [9E9, 9E9, 9E9, 9E9, 9E9, 9E9]];
	VAR jointtarget CDP_2864 := [[11.34, 36.12, 5.45, 0, 48.43, -292.67], [9E9, 9E9, 9E9, 9E9, 9E9, 9E9]];
	VAR jointtarget CDP_2865 := [[11.28, 36.14, 5.42, 0, 48.44, -290.53], [9E9, 9E9, 9E9, 9E9, 9E9, 9E9]];
	VAR jointtarget CDP_2866 := [[11.23, 36.16, 5.38, 0, 48.46, -288.38], [9E9, 9E9, 9E9, 9E9, 9E9, 9E9]];
	VAR jointtarget CDP_2867 := [[11.18, 36.18, 5.35, 0, 48.47, -286.24], [9E9, 9E9, 9E9, 9E9, 9E9, 9E9]];
	VAR jointtarget CDP_2868 := [[11.13, 36.19, 5.33, 0, 48.48, -284.1], [9E9, 9E9, 9E9, 9E9, 9E9, 9E9]];
	VAR jointtarget CDP_2869 := [[11.07, 36.2, 5.31, 0, 48.49, -281.96], [9E9, 9E9, 9E9, 9E9, 9E9, 9E9]];
	VAR jointtarget CDP_2870 := [[11.02, 36.21, 5.29, 0, 48.5, -279.82], [9E9, 9E9, 9E9, 9E9, 9E9, 9E9]];
	VAR jointtarget CDP_2871 := [[10.96, 36.22, 5.28, 0, 48.5, -277.69], [9E9, 9E9, 9E9, 9E9, 9E9, 9E9]];
	VAR jointtarget CDP_2872 := [[10.91, 36.23, 5.27, 0, 48.51, -275.55], [9E9, 9E9, 9E9, 9E9, 9E9, 9E9]];
	VAR jointtarget CDP_2873 := [[10.85, 36.23, 5.26, 0, 48.51, -273.41], [9E9, 9E9, 9E9, 9E9, 9E9, 9E9]];
	VAR jointtarget CDP_2874 := [[10.8, 36.23, 5.26, 0, 48.51, -271.27], [9E9, 9E9, 9E9, 9E9, 9E9, 9E9]];
	VAR jointtarget CDP_2875 := [[10.74, 36.23, 5.26, 0, 48.51, -269.13], [9E9, 9E9, 9E9, 9E9, 9E9, 9E9]];
	VAR jointtarget CDP_2876 := [[10.69, 36.23, 5.27, 0, 48.51, -266.99], [9E9, 9E9, 9E9, 9E9, 9E9, 9E9]];
	VAR jointtarget CDP_2877 := [[10.63, 36.22, 5.27, 0, 48.5, -264.85], [9E9, 9E9, 9E9, 9E9, 9E9, 9E9]];
	VAR jointtarget CDP_2878 := [[10.58, 36.21, 5.29, 0, 48.5, -262.71], [9E9, 9E9, 9E9, 9E9, 9E9, 9E9]];
	VAR jointtarget CDP_2879 := [[10.52, 36.2, 5.3, 0, 48.49, -260.58], [9E9, 9E9, 9E9, 9E9, 9E9, 9E9]];
	VAR jointtarget CDP_2880 := [[9.44, 36, 5.66, 0, 48.34, -260.56], [9E9, 9E9, 9E9, 9E9, 9E9, 9E9]];
	VAR jointtarget CDP_2881 := [[8.36, 35.81, 5.98, 0, 48.21, -261.64], [9E9, 9E9, 9E9, 9E9, 9E9, 9E9]];
	VAR jointtarget CDP_2882 := [[7.27, 35.65, 6.25, 0, 48.1, -262.73], [9E9, 9E9, 9E9, 9E9, 9E9, 9E9]];
	VAR jointtarget CDP_2883 := [[6.17, 35.51, 6.49, 0, 48, -263.83], [9E9, 9E9, 9E9, 9E9, 9E9, 9E9]];
	VAR jointtarget CDP_2884 := [[5.07, 35.4, 6.69, 0, 47.92, -264.93], [9E9, 9E9, 9E9, 9E9, 9E9, 9E9]];
	VAR jointtarget CDP_2885 := [[3.97, 35.3, 6.85, 0, 47.85, -266.03], [9E9, 9E9, 9E9, 9E9, 9E9, 9E9]];
	VAR jointtarget CDP_2886 := [[2.86, 35.23, 6.97, 0, 47.8, -267.14], [9E9, 9E9, 9E9, 9E9, 9E9, 9E9]];
	VAR jointtarget CDP_2887 := [[1.75, 35.18, 7.05, 0, 47.77, -268.25], [9E9, 9E9, 9E9, 9E9, 9E9, 9E9]];
	VAR jointtarget CDP_2888 := [[0.64, 35.16, 7.09, 0, 47.75, -269.36], [9E9, 9E9, 9E9, 9E9, 9E9, 9E9]];
	VAR jointtarget CDP_2889 := [[-0.47, 35.16, 7.09, 0, 47.75, -270.47], [9E9, 9E9, 9E9, 9E9, 9E9, 9E9]];
	VAR jointtarget CDP_2890 := [[-1.58, 35.18, 7.06, 0, 47.76, -271.58], [9E9, 9E9, 9E9, 9E9, 9E9, 9E9]];
	VAR jointtarget CDP_2891 := [[-2.69, 35.22, 6.98, 0, 47.79, -272.69], [9E9, 9E9, 9E9, 9E9, 9E9, 9E9]];
	VAR jointtarget CDP_2892 := [[-3.8, 35.29, 6.87, 0, 47.84, -273.8], [9E9, 9E9, 9E9, 9E9, 9E9, 9E9]];
	VAR jointtarget CDP_2893 := [[-4.9, 35.38, 6.72, 0, 47.9, -274.9], [9E9, 9E9, 9E9, 9E9, 9E9, 9E9]];
	VAR jointtarget CDP_2894 := [[-6, 35.49, 6.52, 0, 47.98, -276], [9E9, 9E9, 9E9, 9E9, 9E9, 9E9]];
	VAR jointtarget CDP_2895 := [[-7.1, 35.63, 6.29, 0, 48.08, -277.1], [9E9, 9E9, 9E9, 9E9, 9E9, 9E9]];
	VAR jointtarget CDP_2896 := [[-8.19, 35.79, 6.02, 0, 48.19, -278.19], [9E9, 9E9, 9E9, 9E9, 9E9, 9E9]];
	VAR jointtarget CDP_2897 := [[-9.28, 35.97, 5.71, 0, 48.32, -279.28], [9E9, 9E9, 9E9, 9E9, 9E9, 9E9]];
	VAR jointtarget CDP_2898 := [[-10.36, 36.17, 5.36, 0, 48.47, -280.36], [9E9, 9E9, 9E9, 9E9, 9E9, 9E9]];
	VAR jointtarget CDP_2899 := [[-11.43, 36.4, 4.97, 0, 48.63, -281.43], [9E9, 9E9, 9E9, 9E9, 9E9, 9E9]];
	VAR jointtarget CDP_2900 := [[-11.44, 36.4, 4.97, 0, 48.63, -281.78], [9E9, 9E9, 9E9, 9E9, 9E9, 9E9]];
	VAR jointtarget CDP_2901 := [[-11.46, 36.41, 4.96, 0, 48.63, -282.45], [9E9, 9E9, 9E9, 9E9, 9E9, 9E9]];
	VAR jointtarget CDP_2902 := [[-11.48, 36.41, 4.95, 0, 48.64, -283.13], [9E9, 9E9, 9E9, 9E9, 9E9, 9E9]];
	VAR jointtarget CDP_2903 := [[-11.49, 36.41, 4.95, 0, 48.64, -283.81], [9E9, 9E9, 9E9, 9E9, 9E9, 9E9]];
	VAR jointtarget CDP_2904 := [[-11.51, 36.42, 4.94, 0, 48.64, -284.49], [9E9, 9E9, 9E9, 9E9, 9E9, 9E9]];
	VAR jointtarget CDP_2905 := [[-11.53, 36.42, 4.93, 0, 48.65, -285.17], [9E9, 9E9, 9E9, 9E9, 9E9, 9E9]];
	VAR jointtarget CDP_2906 := [[-11.54, 36.43, 4.92, 0, 48.65, -285.84], [9E9, 9E9, 9E9, 9E9, 9E9, 9E9]];
	VAR jointtarget CDP_2907 := [[-11.56, 36.43, 4.91, 0, 48.65, -286.52], [9E9, 9E9, 9E9, 9E9, 9E9, 9E9]];
	VAR jointtarget CDP_2908 := [[-11.57, 36.44, 4.9, 0, 48.66, -287.2], [9E9, 9E9, 9E9, 9E9, 9E9, 9E9]];
	VAR jointtarget CDP_2909 := [[-11.59, 36.44, 4.89, 0, 48.66, -287.88], [9E9, 9E9, 9E9, 9E9, 9E9, 9E9]];
	VAR jointtarget CDP_2910 := [[-11.6, 36.45, 4.88, 0, 48.67, -288.56], [9E9, 9E9, 9E9, 9E9, 9E9, 9E9]];
	VAR jointtarget CDP_2911 := [[-11.62, 36.46, 4.87, 0, 48.67, -289.23], [9E9, 9E9, 9E9, 9E9, 9E9, 9E9]];
	VAR jointtarget CDP_2912 := [[-11.64, 36.46, 4.86, 0, 48.67, -289.91], [9E9, 9E9, 9E9, 9E9, 9E9, 9E9]];
	VAR jointtarget CDP_2913 := [[-11.65, 36.47, 4.85, 0, 48.68, -290.59], [9E9, 9E9, 9E9, 9E9, 9E9, 9E9]];
	VAR jointtarget CDP_2914 := [[-11.67, 36.48, 4.84, 0, 48.68, -291.27], [9E9, 9E9, 9E9, 9E9, 9E9, 9E9]];
	VAR jointtarget CDP_2915 := [[-11.68, 36.48, 4.83, 0, 48.69, -291.94], [9E9, 9E9, 9E9, 9E9, 9E9, 9E9]];
	VAR jointtarget CDP_2916 := [[-11.7, 36.49, 4.82, 0, 48.69, -292.62], [9E9, 9E9, 9E9, 9E9, 9E9, 9E9]];
	VAR jointtarget CDP_2917 := [[-11.71, 36.5, 4.8, 0, 48.7, -293.3], [9E9, 9E9, 9E9, 9E9, 9E9, 9E9]];
